C01810=1045.452,114.754,411.757,170.471,36.700,156.909
C01811=1045.446,114.505,411.777,170.469,36.699,156.908
C01812=1045.440,114.256,411.797,170.467,36.698,156.908
C01813=1045.434,114.007,411.817,170.464,36.696,156.908
C01814=1045.428,113.757,411.838,170.463,36.695,156.908
C01815=1045.422,113.509,411.858,170.461,36.693,156.907
C01816=1045.416,113.260,411.878,170.459,36.692,156.907
C01817=1045.410,113.010,411.898,170.458,36.690,156.907
C01818=1045.404,112.761,411.918,170.456,36.689,156.906
C01819=1045.398,112.512,411.937,170.453,36.687,156.906
C01820=1045.391,112.263,411.957,170.451,36.686,156.906
C01821=1045.385,112.014,411.977,170.450,36.684,156.906
C01822=1045.379,111.765,411.997,170.448,36.683,156.905
C01823=1045.373,111.515,412.018,170.446,36.681,156.905
C01824=1045.367,111.267,412.038,170.444,36.680,156.905
C01825=1045.361,111.018,412.058,170.442,36.679,156.904
C01826=1045.354,110.768,412.078,170.440,36.677,156.904
C01827=1045.348,110.519,412.097,170.438,36.676,156.904
C01828=1045.342,110.270,412.117,170.437,36.674,156.904
C01829=1045.336,110.020,412.137,170.435,36.673,156.903
C01830=1045.328,109.735,412.160,170.432,36.671,156.903
C01831=1045.322,109.449,412.183,170.430,36.669,156.903
C01832=1045.314,109.163,412.205,170.428,36.668,156.902
C01833=1045.308,108.877,412.228,170.426,36.666,156.902
C01834=1045.301,108.627,412.248,170.424,36.665,156.902
C01835=1045.295,108.379,412.268,170.423,36.664,156.902
C01836=1045.288,108.130,412.287,170.420,36.662,156.901
C01837=1045.283,107.881,412.307,170.418,36.661,156.901
C01838=1045.276,107.631,412.327,170.416,36.659,156.901
C01839=1045.270,107.382,412.347,170.415,36.658,156.900
C01840=1045.264,107.133,412.366,170.413,36.656,156.900
C01841=1045.258,106.883,412.387,170.411,36.655,156.900
C01842=1045.251,106.635,412.406,170.409,36.653,156.900
C01843=1045.245,106.386,412.425,170.407,36.652,156.899
C01844=1045.239,106.137,412.445,170.405,36.651,156.899
C01845=1045.233,105.887,412.466,170.403,36.650,156.899
C01846=1045.227,105.638,412.485,170.402,36.648,156.898
C01847=1045.221,105.389,412.505,170.399,36.646,156.898
C01848=1045.214,105.140,412.524,170.397,36.645,156.898
C01849=1045.208,104.890,412.544,170.396,36.643,156.898
C01850=1045.202,104.642,412.564,170.394,36.642,156.897
C01851=1045.196,104.392,412.583,170.392,36.641,156.897
C01852=1045.190,104.143,412.603,170.391,36.639,156.897
C01853=1045.184,103.894,412.623,170.388,36.638,156.896
C01854=1045.177,103.645,412.642,170.386,36.637,156.896
C01855=1045.171,103.396,412.662,170.384,36.635,156.896
C01856=1045.166,103.146,412.681,170.383,36.633,156.896
C01857=1045.160,102.898,412.701,170.381,36.632,156.895
C01858=1045.154,102.649,412.721,170.379,36.630,156.895
C01859=1045.147,102.399,412.741,170.377,36.629,156.895
C01860=1045.141,102.150,412.760,170.375,36.628,156.895
C01861=1045.135,101.901,412.779,170.373,36.626,156.894
C01862=1045.129,101.652,412.799,170.372,36.625,156.894
C01863=1045.123,101.402,412.818,170.370,36.624,156.894
C01864=1045.117,101.154,412.838,170.368,36.622,156.893
C01865=1045.110,100.904,412.857,170.366,36.620,156.893
C01866=1045.104,100.655,412.877,170.364,36.619,156.893
C01867=1045.098,100.406,412.897,170.362,36.618,156.893
C01868=1045.092,100.157,412.916,170.360,36.616,156.892
C01869=1045.086,99.908,412.935,170.359,36.615,156.892
C01870=1045.079,99.658,412.956,170.357,36.614,156.892
C01871=1045.073,99.409,412.974,170.354,36.612,156.892
C01872=1045.067,99.160,412.993,170.353,36.611,156.891
C01873=1045.061,98.911,413.013,170.351,36.609,156.891
C01874=1045.055,98.662,413.032,170.349,36.608,156.891
C01875=1045.048,98.413,413.051,170.348,36.607,156.890
C01876=1045.042,98.163,413.071,170.346,36.605,156.890
C01877=1045.035,97.914,413.090,170.343,36.604,156.890
C01878=1045.029,97.665,413.110,170.341,36.602,156.890
C01879=1045.024,97.416,413.129,170.340,36.601,156.889
C01880=1045.017,97.167,413.148,170.338,36.600,156.889
C01881=1045.011,96.918,413.167,170.336,36.599,156.889
C01882=1045.005,96.669,413.186,170.335,36.597,156.889
C01883=1044.999,96.418,413.206,170.332,36.596,156.888
C01884=1044.992,96.170,413.225,170.330,36.594,156.888
C01885=1044.986,95.921,413.244,170.329,36.593,156.888
C01886=1044.980,95.671,413.263,170.327,36.591,156.887
C01887=1044.974,95.423,413.283,170.325,36.590,156.887
C01888=1044.967,95.173,413.302,170.324,36.589,156.887
C01889=1044.962,94.924,413.321,170.321,36.587,156.887
C01890=1044.956,94.675,413.340,170.319,36.586,156.886
C01891=1044.949,94.426,413.359,170.318,36.584,156.886
C01892=1044.943,94.176,413.379,170.316,36.583,156.886
C01893=1044.937,93.927,413.398,170.314,36.582,156.886
C01894=1044.930,93.642,413.420,170.312,36.580,156.885
C01895=1044.923,93.355,413.441,170.309,36.579,156.885
C01896=1044.916,93.069,413.464,170.307,36.577,156.885
C01897=1044.909,92.783,413.486,170.305,36.575,156.884
C01898=1044.902,92.534,413.505,170.304,36.574,156.884
C01899=1044.896,92.285,413.525,170.302,36.572,156.884
C01900=1044.890,92.036,413.543,170.300,36.571,156.884
C01901=1044.884,91.787,413.562,170.298,36.569,156.883
C01902=1044.878,91.538,413.581,170.296,36.568,156.883
C01903=1044.872,91.288,413.600,170.294,36.567,156.883
C01904=1044.866,91.039,413.619,170.293,36.566,156.883
C01905=1044.860,90.790,413.639,170.291,36.564,156.882
C01906=1044.853,90.541,413.658,170.289,36.562,156.882
C01907=1044.848,90.292,413.677,170.287,36.561,156.882
C01908=1044.841,90.043,413.695,170.285,36.560,156.881
C01909=1044.835,89.793,413.714,170.283,36.559,156.881
C01910=1044.829,89.544,413.733,170.282,36.557,156.881
C01911=1044.822,89.294,413.752,170.280,36.556,156.881
C01912=1044.816,89.045,413.771,170.278,36.554,156.880
C01913=1044.809,88.796,413.790,170.276,36.553,156.880
C01914=1044.803,88.546,413.809,170.274,36.552,156.880
C01915=1044.797,88.297,413.828,170.272,36.551,156.880
C01916=1044.791,88.048,413.846,170.271,36.549,156.879
C01917=1044.784,87.799,413.865,170.269,36.548,156.879
C01918=1044.779,87.550,413.884,170.267,36.546,156.879
C01919=1044.772,87.301,413.903,170.265,36.545,156.879
C01920=1044.766,87.051,413.921,170.263,36.544,156.878
C01921=1044.759,86.802,413.940,170.261,36.543,156.878
C01922=1044.754,86.553,413.959,170.259,36.541,156.878
C01923=1044.747,86.304,413.978,170.258,36.540,156.878
C01924=1044.741,86.055,413.997,170.256,36.538,156.877
C01925=1044.734,85.805,414.015,170.254,36.537,156.877
C01926=1044.729,85.556,414.034,170.252,36.536,156.877
C01927=1044.722,85.307,414.053,170.250,36.534,156.877
C01928=1044.716,85.058,414.072,170.248,36.533,156.876
C01929=1044.709,84.809,414.090,170.247,36.532,156.876
C01930=1044.703,84.560,414.109,170.245,36.530,156.876
C01931=1044.697,84.310,414.128,170.243,36.529,156.876
C01932=1044.691,84.061,414.147,170.242,36.528,156.875
C01933=1044.684,83.812,414.166,170.239,36.526,156.875
C01934=1044.678,83.562,414.184,170.237,36.525,156.875
C01935=1044.673,83.313,414.203,170.236,36.524,156.875
C01936=1044.666,83.064,414.221,170.234,36.522,156.874
C01937=1044.660,82.815,414.240,170.232,36.521,156.874
C01938=1044.654,82.566,414.258,170.231,36.519,156.874
C01939=1044.647,82.317,414.277,170.228,36.518,156.873
C01940=1044.642,82.067,414.296,170.226,36.517,156.873
C01941=1044.636,81.818,414.314,170.225,36.516,156.873
C01942=1044.629,81.569,414.333,170.223,36.514,156.873
C01943=1044.623,81.320,414.351,170.221,36.513,156.872
C01944=1044.616,81.070,414.370,170.220,36.511,156.872
C01945=1044.611,80.821,414.389,170.218,36.510,156.872
C01946=1044.604,80.572,414.408,170.215,36.509,156.872
C01947=1044.598,80.322,414.426,170.214,36.507,156.871
C01948=1044.592,80.074,414.444,170.212,36.506,156.871
C01949=1044.586,79.825,414.463,170.210,36.504,156.871
C01950=1044.580,79.575,414.482,170.209,36.503,156.871
C01951=1044.574,79.325,414.500,170.207,36.502,156.870
C01952=1044.568,79.076,414.519,170.204,36.500,156.870
C01953=1044.561,78.827,414.537,170.203,36.499,156.870
C01954=1044.555,78.578,414.556,170.201,36.497,156.870
C01955=1044.549,78.328,414.574,170.199,36.496,156.869
C01956=1044.543,78.080,414.592,170.198,36.495,156.869
C01957=1044.536,77.831,414.611,170.196,36.494,156.869
C01958=1044.529,77.544,414.632,170.194,36.492,156.869
C01959=1044.523,77.258,414.653,170.191,36.491,156.868
C01960=1044.515,76.972,414.674,170.189,36.489,156.868
C01961=1044.508,76.686,414.696,170.187,36.487,156.868
C01962=1044.502,76.437,414.714,170.186,36.486,156.867
C01963=1044.496,76.188,414.732,170.184,36.485,156.867
C01964=1044.490,75.939,414.751,170.182,36.484,156.867
C01965=1044.483,75.689,414.768,170.180,36.482,156.867
C01966=1044.476,75.440,414.787,170.178,36.481,156.866
C01967=1044.470,75.191,414.805,170.176,36.479,156.866
C01968=1044.464,74.941,414.823,170.174,36.478,156.866
C01969=1044.457,74.692,414.842,170.173,36.477,156.866
C01970=1044.452,74.443,414.859,170.171,36.476,156.865
C01971=1044.445,74.194,414.878,170.169,36.474,156.865
C01972=1044.439,73.945,414.897,170.167,36.473,156.865
C01973=1044.433,73.695,414.915,170.165,36.472,156.865
C01974=1044.426,73.446,414.933,170.163,36.471,156.864
C01975=1044.420,73.196,414.951,170.162,36.469,156.864
C01976=1044.415,72.948,414.969,170.160,36.467,156.864
C01977=1044.408,72.698,414.987,170.158,36.466,156.864
C01978=1044.402,72.449,415.006,170.157,36.465,156.863
C01979=1044.395,72.199,415.023,170.154,36.464,156.863
C01980=1044.389,71.950,415.042,170.152,36.462,156.863
C01981=1044.383,71.701,415.060,170.151,36.461,156.863
C01982=1044.377,71.452,415.078,170.149,36.460,156.862
C01983=1044.371,71.202,415.096,170.147,36.459,156.862
C01984=1044.364,70.953,415.115,170.146,36.457,156.862
C01985=1044.359,70.704,415.132,170.143,36.455,156.862
C01986=1044.352,70.455,415.151,170.141,36.454,156.861
C01987=1044.346,70.205,415.169,170.140,36.453,156.861
C01988=1044.339,69.956,415.186,170.138,36.452,156.861
C01989=1044.333,69.707,415.205,170.136,36.450,156.861
C01990=1044.327,69.458,415.223,170.135,36.449,156.860
C01991=1044.321,69.209,415.241,170.133,36.448,156.860
C01992=1044.315,68.959,415.259,170.130,36.447,156.860
C01993=1044.308,68.709,415.276,170.129,36.445,156.860
C01994=1044.302,68.461,415.295,170.127,36.444,156.860
C01995=1044.296,68.211,415.313,170.125,36.443,156.859
C01996=1044.290,67.962,415.331,170.124,36.442,156.859
C01997=1044.283,67.713,415.349,170.122,36.440,156.859
C01998=1044.277,67.464,415.366,170.120,36.438,156.858
C01999=1044.271,67.214,415.384,170.117,36.437,156.858
C02000=1044.265,66.965,415.403,170.116,36.436,156.858
C02001=1044.258,66.715,415.420,170.114,36.435,156.858
C02002=1044.252,66.466,415.438,170.112,36.433,156.857
C02003=1044.246,66.217,415.456,170.111,36.432,156.857
C02004=1044.240,65.968,415.474,170.109,36.431,156.857
C02005=1044.233,65.718,415.492,170.107,36.430,156.857
C02006=1044.227,65.469,415.509,170.105,36.428,156.857
C02007=1044.221,65.220,415.528,170.103,36.427,156.856
C02008=1044.214,64.970,415.545,170.101,36.426,156.856
C02009=1044.209,64.721,415.563,170.100,36.425,156.856
C02010=1044.202,64.472,415.581,170.098,36.423,156.856
C02011=1044.195,64.223,415.599,170.096,36.422,156.855
C02012=1044.189,63.973,415.617,170.095,36.421,156.855
C02013=1044.184,63.724,415.634,170.093,36.420,156.855
C02014=1044.177,63.475,415.652,170.090,36.418,156.855
C02015=1044.170,63.225,415.669,170.088,36.417,156.854
C02016=1044.164,62.976,415.687,170.087,36.416,156.854
C02017=1044.157,62.727,415.705,170.085,36.415,156.854
C02018=1044.151,62.478,415.722,170.083,36.413,156.854
C02019=1044.144,62.228,415.740,170.082,36.412,156.853
C02020=1044.139,61.979,415.757,170.080,36.411,156.853
C02021=1044.132,61.730,415.775,170.078,36.410,156.853
C02022=1044.124,61.443,415.795,170.075,36.408,156.853
C02023=1044.117,61.157,415.815,170.073,36.407,156.853
C02024=1044.110,60.871,415.835,170.071,36.406,156.852
C02025=1044.103,60.585,415.855,170.069,36.404,156.852
C02026=1044.096,60.335,415.873,170.068,36.403,156.852
C02027=1044.090,60.085,415.890,170.066,36.402,156.852
C02028=1044.083,59.837,415.908,170.063,36.401,156.851
C02029=1044.076,59.588,415.926,170.062,36.399,156.851
C02030=1044.070,59.338,415.943,170.060,36.398,156.851
C02031=1044.064,59.089,415.960,170.058,36.397,156.851
C02032=1044.058,58.840,415.978,170.056,36.396,156.850
C02033=1044.051,58.590,415.996,170.055,36.394,156.850
C02034=1044.045,58.342,416.013,170.053,36.393,156.850
C02035=1044.039,58.092,416.031,170.051,36.392,156.850
C02036=1044.032,57.843,416.048,170.049,36.391,156.849
C02037=1044.026,57.593,416.066,170.047,36.389,156.849
C02038=1044.019,57.344,416.083,170.045,36.388,156.849
C02039=1044.013,57.095,416.100,170.043,36.387,156.849
C02040=1044.007,56.845,416.118,170.042,36.386,156.849
C02041=1044.000,56.596,416.135,170.040,36.385,156.848
C02042=1043.995,56.346,416.152,170.038,36.384,156.848
C02043=1043.988,56.097,416.169,170.037,36.382,156.848
C02044=1043.982,55.848,416.186,170.034,36.381,156.848
C02045=1043.976,55.598,416.204,170.032,36.380,156.848
C02046=1043.969,55.349,416.222,170.031,36.379,156.847
C02047=1043.963,55.100,416.239,170.029,36.377,156.847
C02048=1043.957,54.851,416.256,170.027,36.376,156.847
C02049=1043.950,54.602,416.273,170.025,36.375,156.847
C02050=1043.944,54.352,416.291,170.024,36.373,156.846
C02051=1043.937,54.103,416.309,170.021,36.372,156.846
C02052=1043.931,53.854,416.326,170.019,36.371,156.846
C02053=1043.925,53.604,416.343,170.018,36.370,156.846
C02054=1043.919,53.355,416.360,170.016,36.368,156.845
C02055=1043.913,53.105,416.378,170.014,36.367,156.845
C02056=1043.907,52.856,416.395,170.012,36.366,156.845
C02057=1043.900,52.607,416.412,170.011,36.365,156.845
C02058=1043.894,52.358,416.430,170.009,36.363,156.844
C02059=1043.888,52.108,416.446,170.006,36.362,156.844
C02060=1043.881,51.859,416.463,170.005,36.361,156.844
C02061=1043.875,51.609,416.481,170.003,36.360,156.844
C02062=1043.869,51.361,416.498,170.001,36.358,156.844
C02063=1043.862,51.111,416.515,170.000,36.357,156.843
C02064=1043.857,50.862,416.532,169.998,36.356,156.843
C02065=1043.850,50.612,416.550,169.996,36.355,156.843
C02066=1043.844,50.363,416.567,169.993,36.353,156.843
C02067=1043.838,50.114,416.585,169.992,36.352,156.842
C02068=1043.831,49.865,416.602,169.990,36.351,156.842
C02069=1043.825,49.615,416.618,169.988,36.349,156.842
C02070=1043.819,49.366,416.636,169.987,36.348,156.842
C02071=1043.813,49.116,416.653,169.985,36.347,156.841
C02072=1043.807,48.867,416.671,169.983,36.346,156.841
C02073=1043.800,48.617,416.687,169.981,36.344,156.841
C02074=1043.794,48.369,416.704,169.979,36.343,156.841
C02075=1043.788,48.119,416.722,169.977,36.342,156.840
C02076=1043.782,47.869,416.738,169.975,36.341,156.840
C02077=1043.775,47.620,416.756,169.974,36.339,156.840
C02078=1043.770,47.371,416.773,169.972,36.338,156.840
C02079=1043.763,47.121,416.790,169.970,36.337,156.840
C02080=1043.757,46.872,416.807,169.969,36.336,156.839
C02081=1043.751,46.624,416.824,169.966,36.334,156.839
C02082=1043.745,46.373,416.841,169.964,36.333,156.839
C02083=1043.739,46.124,416.858,169.963,36.332,156.839
C02084=1043.732,45.875,416.875,169.961,36.330,156.838
C02085=1043.727,45.625,416.892,169.959,36.329,156.838
C02086=1043.720,45.339,416.912,169.957,36.328,156.838
C02087=1043.712,45.052,416.932,169.955,36.326,156.838
C02088=1043.705,44.766,416.950,169.952,36.325,156.837
C02089=1043.698,44.480,416.970,169.950,36.323,156.837
C02090=1043.692,44.230,416.988,169.949,36.322,156.837
C02091=1043.686,43.981,417.005,169.947,36.321,156.837
C02092=1043.679,43.731,417.022,169.945,36.320,156.836
C02093=1043.674,43.482,417.039,169.944,36.318,156.836
C02094=1043.668,43.233,417.056,169.942,36.317,156.836
C02095=1043.661,42.983,417.072,169.940,36.316,156.836
C02096=1043.655,42.734,417.089,169.937,36.315,156.835
C02097=1043.648,42.484,417.106,169.936,36.313,156.835
C02098=1043.642,42.235,417.123,169.934,36.312,156.835
C02099=1043.636,41.986,417.139,169.932,36.311,156.835
C02100=1043.629,41.737,417.157,169.930,36.309,156.835
C02101=1043.623,41.487,417.173,169.929,36.308,156.834
C02102=1043.616,41.238,417.190,169.927,36.307,156.834
C02103=1043.610,40.989,417.206,169.925,36.306,156.834
C02104=1043.604,40.739,417.223,169.923,36.305,156.834
C02105=1043.598,40.490,417.240,169.921,36.304,156.833
C02106=1043.592,40.240,417.256,169.919,36.302,156.833
C02107=1043.586,39.991,417.274,169.917,36.301,156.833
C02108=1043.580,39.741,417.290,169.916,36.300,156.833
C02109=1043.573,39.493,417.307,169.914,36.299,156.833
C02110=1043.567,39.243,417.324,169.912,36.297,156.832
C02111=1043.561,38.993,417.340,169.909,36.296,156.832
C02112=1043.555,38.744,417.357,169.908,36.295,156.832
C02113=1043.549,38.495,417.374,169.906,36.294,156.832
C02114=1043.542,38.245,417.390,169.904,36.293,156.832
C02115=1043.536,37.996,417.407,169.903,36.292,156.831
C02116=1043.530,37.747,417.423,169.901,36.290,156.831
C02117=1043.523,37.497,417.440,169.899,36.289,156.831
C02118=1043.517,37.248,417.457,169.897,36.288,156.831
C02119=1043.510,36.998,417.474,169.896,36.287,156.830
C02120=1043.505,36.749,417.490,169.893,36.285,156.830
C02121=1043.498,36.500,417.506,169.891,36.285,156.830
C02122=1043.491,36.250,417.523,169.889,36.283,156.830
C02123=1043.485,36.001,417.539,169.888,36.282,156.830
C02124=1043.479,35.752,417.555,169.886,36.281,156.829
C02125=1043.472,35.502,417.573,169.884,36.280,156.829
C02126=1043.466,35.253,417.589,169.882,36.279,156.829
C02127=1043.460,35.004,417.605,169.880,36.278,156.829
C02128=1043.453,34.754,417.621,169.878,36.276,156.829
C02129=1043.447,34.504,417.638,169.876,36.275,156.828
C02130=1043.441,34.256,417.654,169.874,36.274,156.828
C02131=1043.435,34.006,417.671,169.872,36.273,156.828
C02132=1043.428,33.757,417.687,169.871,36.272,156.828
C02133=1043.422,33.507,417.703,169.869,36.271,156.827
C02134=1043.416,33.258,417.719,169.867,36.269,156.827
C02135=1043.409,33.009,417.737,169.865,36.268,156.827
C02136=1043.403,32.759,417.753,169.864,36.267,156.827
C02137=1043.397,32.510,417.769,169.861,36.266,156.827
C02138=1043.390,32.261,417.785,169.859,36.265,156.826
C02139=1043.384,32.011,417.801,169.857,36.264,156.826
C02140=1043.378,31.761,417.818,169.856,36.262,156.826
C02141=1043.371,31.513,417.835,169.854,36.261,156.826
C02142=1043.365,31.263,417.851,169.852,36.260,156.825
C02143=1043.358,31.014,417.867,169.850,36.259,156.825
C02144=1043.352,30.764,417.883,169.849,36.258,156.825
C02145=1043.346,30.515,417.899,169.846,36.257,156.825
C02146=1043.340,30.266,417.916,169.844,36.255,156.825
C02147=1043.334,30.015,417.932,169.842,36.254,156.824
C02148=1043.327,29.766,417.948,169.840,36.253,156.824
C02149=1043.321,29.517,417.964,169.839,36.252,156.824
C02150=1043.314,29.231,417.983,169.837,36.251,156.824
C02151=1043.307,28.944,418.002,169.835,36.249,156.824
C02152=1043.300,28.657,418.020,169.833,36.248,156.823
C02153=1043.292,28.370,418.039,169.830,36.246,156.823
C02154=1043.286,28.121,418.055,169.828,36.245,156.823
C02155=1043.279,27.872,418.071,169.826,36.244,156.823
C02156=1043.273,27.623,418.087,169.824,36.243,156.823
C02157=1043.267,27.373,418.103,169.822,36.242,156.822
C02158=1043.260,27.124,418.120,169.821,36.241,156.822
C02159=1043.254,26.874,418.136,169.819,36.240,156.822
C02160=1043.248,26.625,418.152,169.817,36.239,156.822
C02161=1043.242,26.376,418.168,169.815,36.237,156.821
C02162=1043.236,26.127,418.184,169.813,36.236,156.821
C02163=1043.228,25.877,418.200,169.811,36.236,156.821
C02164=1043.222,25.627,418.216,169.809,36.234,156.821
C02165=1043.216,25.378,418.232,169.807,36.233,156.821
C02166=1043.210,25.128,418.247,169.805,36.232,156.821
C02167=1043.204,24.879,418.264,169.804,36.231,156.820
C02168=1043.197,24.629,418.280,169.802,36.230,156.820
C02169=1043.191,24.380,418.296,169.800,36.228,156.820
C02170=1043.184,24.131,418.312,169.798,36.228,156.820
C02171=1043.178,23.882,418.328,169.795,36.227,156.820
C02172=1043.172,23.632,418.344,169.794,36.225,156.819
C02173=1043.166,23.383,418.359,169.792,36.224,156.819
C02174=1043.159,23.133,418.376,169.790,36.223,156.819
C02175=1043.153,22.884,418.391,169.788,36.222,156.819
C02176=1043.147,22.634,418.408,169.786,36.221,156.818
C02177=1043.140,22.385,418.423,169.785,36.219,156.818
C02178=1043.134,22.136,418.440,169.783,36.219,156.818
C02179=1043.128,21.886,418.454,169.781,36.218,156.818
C02180=1043.122,21.637,418.471,169.778,36.216,156.818
C02181=1043.115,21.388,418.486,169.776,36.215,156.817
C02182=1043.109,21.138,418.503,169.775,36.214,156.817
C02183=1043.103,20.888,418.519,169.773,36.213,156.817
C02184=1043.096,20.639,418.534,169.771,36.212,156.817
C02185=1043.090,20.389,418.550,169.769,36.211,156.817
C02186=1043.084,20.140,418.566,169.767,36.210,156.817
C02187=1043.078,19.890,418.582,169.766,36.209,156.816
C02188=1043.071,19.641,418.597,169.764,36.207,156.816
C02189=1043.065,19.392,418.614,169.762,36.207,156.816
C02190=1043.059,19.143,418.629,169.759,36.205,156.816
C02191=1043.052,18.893,418.644,169.757,36.204,156.815
C02192=1043.046,18.644,418.660,169.755,36.203,156.815
C02193=1043.039,18.394,418.677,169.754,36.202,156.815
C02194=1043.033,18.144,418.692,169.752,36.201,156.815
C02195=1043.027,17.895,418.708,169.750,36.200,156.815
C02196=1043.020,17.646,418.723,169.748,36.199,156.815
C02197=1043.014,17.396,418.739,169.746,36.198,156.814
C02198=1043.008,17.147,418.755,169.745,36.197,156.814
C02199=1043.002,16.897,418.770,169.742,36.196,156.814
C02200=1042.995,16.648,418.786,169.740,36.194,156.814
C02201=1042.989,16.399,418.801,169.738,36.194,156.814
C02202=1042.983,16.149,418.817,169.736,36.193,156.813
C02203=1042.976,15.900,418.833,169.734,36.191,156.813
C02204=1042.970,15.650,418.848,169.733,36.190,156.813
C02205=1042.964,15.401,418.864,169.731,36.189,156.813
C02206=1042.957,15.152,418.880,169.729,36.188,156.813
C02207=1042.952,14.902,418.895,169.727,36.187,156.812
C02208=1042.945,14.653,418.911,169.725,36.186,156.812
C02209=1042.938,14.403,418.926,169.722,36.185,156.812
C02210=1042.933,14.154,418.942,169.721,36.184,156.812
C02211=1042.926,13.904,418.957,169.719,36.183,156.812
C02212=1042.919,13.655,418.973,169.717,36.182,156.811
C02213=1042.913,13.406,418.987,169.715,36.181,156.811
C02214=1042.906,13.120,419.005,169.713,36.180,156.811
C02215=1042.898,12.835,419.023,169.711,36.178,156.811
C02216=1042.891,12.550,419.041,169.709,36.177,156.811
C02217=1042.884,12.265,419.059,169.707,36.176,156.811
C02218=1042.877,12.015,419.074,169.704,36.175,156.810
C02219=1042.871,11.765,419.089,169.702,36.174,156.810
C02220=1042.864,11.516,419.104,169.700,36.173,156.810
C02221=1042.858,11.267,419.119,169.698,36.172,156.810
C02222=1042.851,11.017,419.135,169.696,36.171,156.810
C02223=1042.845,10.768,419.150,169.694,36.170,156.809
C02224=1042.839,10.518,419.165,169.692,36.169,156.809
C02225=1042.832,10.269,419.181,169.691,36.168,156.809
C02226=1042.826,10.019,419.196,169.689,36.167,156.809
C02227=1042.819,9.770,419.212,169.687,36.166,156.809
C02228=1042.813,9.520,419.227,169.685,36.165,156.809
C02229=1042.807,9.271,419.242,169.682,36.164,156.808
C02230=1042.800,9.022,419.257,169.680,36.163,156.808
C02231=1042.793,8.772,419.272,169.678,36.162,156.808
C02232=1042.788,8.522,419.288,169.676,36.161,156.808
C02233=1042.781,8.273,419.303,169.675,36.160,156.808
C02234=1042.775,8.023,419.318,169.673,36.159,156.808
C02235=1042.768,7.774,419.333,169.671,36.158,156.807
C02236=1042.762,7.524,419.348,169.669,36.157,156.807
C02237=1042.755,7.275,419.364,169.667,36.156,156.807
C02238=1042.750,7.026,419.378,169.665,36.155,156.807
C02239=1042.743,6.776,419.393,169.662,36.154,156.807
C02240=1042.736,6.527,419.409,169.660,36.153,156.807
C02241=1042.730,6.278,419.424,169.659,36.152,156.806
C02242=1042.724,6.028,419.440,169.657,36.151,156.806
C02243=1042.718,5.778,419.455,169.655,36.150,156.806
C02244=1042.712,5.528,419.469,169.653,36.149,156.806
C02245=1042.705,5.279,419.485,169.651,36.148,156.806
C02246=1042.699,5.030,419.500,169.649,36.147,156.805
C02247=1042.693,4.781,419.515,169.647,36.146,156.805
C02248=1042.686,4.531,419.530,169.645,36.145,156.805
C02249=1042.680,4.282,419.545,169.643,36.144,156.805
C02250=1042.673,4.033,419.560,169.641,36.143,156.805
C02251=1042.667,3.783,419.575,169.639,36.142,156.805
C02252=1042.661,3.533,419.590,169.637,36.141,156.804
C02253=1042.655,3.283,419.606,169.635,36.140,156.804
C02254=1042.649,3.034,419.620,169.633,36.139,156.804
C02255=1042.642,2.785,419.636,169.631,36.138,156.804
C02256=1042.636,2.536,419.651,169.629,36.137,156.804
C02257=1042.630,2.286,419.666,169.627,36.136,156.803
C02258=1042.623,2.036,419.681,169.625,36.135,156.803
C02259=1042.617,1.787,419.696,169.624,36.134,156.803
C02260=1042.611,1.538,419.710,169.622,36.133,156.803
C02261=1042.605,1.288,419.725,169.619,36.132,156.803
C02262=1042.598,1.038,419.740,169.617,36.131,156.803
C02263=1042.592,0.789,419.755,169.615,36.130,156.802
C02264=1042.585,0.540,419.771,169.613,36.129,156.802
C02265=1042.580,0.291,419.785,169.611,36.128,156.802
C02266=1042.573,0.041,419.800,169.609,36.127,156.802
C02267=1042.567,-0.209,419.815,169.607,36.126,156.802
C02268=1042.560,-0.458,419.830,169.605,36.125,156.802
C02269=1042.555,-0.707,419.845,169.604,36.124,156.801
C02270=1042.548,-0.957,419.860,169.602,36.123,156.801
C02271=1042.543,-1.207,419.875,169.599,36.121,156.801
C02272=1042.536,-1.457,419.890,169.597,36.121,156.801
C02273=1042.530,-1.705,419.905,169.595,36.120,156.801
C02274=1042.524,-1.955,419.920,169.593,36.119,156.801
C02275=1042.518,-2.205,419.935,169.591,36.118,156.800
C02276=1042.511,-2.454,419.950,169.589,36.117,156.800
C02277=1042.505,-2.703,419.964,169.587,36.116,156.800
C02278=1042.498,-2.987,419.981,169.585,36.114,156.800
C02279=1042.490,-3.270,419.998,169.583,36.113,156.799
C02280=1042.484,-3.554,420.015,169.581,36.112,156.799
C02281=1042.477,-3.838,420.031,169.578,36.111,156.799
C02282=1042.470,-4.087,420.046,169.576,36.110,156.799
C02283=1042.464,-4.336,420.060,169.574,36.109,156.799
C02284=1042.458,-4.586,420.075,169.572,36.108,156.799
C02285=1042.451,-4.835,420.090,169.570,36.108,156.799
C02286=1042.444,-5.085,420.104,169.568,36.106,156.798
C02287=1042.439,-5.334,420.118,169.566,36.106,156.798
C02288=1042.432,-5.584,420.133,169.564,36.105,156.798
C02289=1042.425,-5.833,420.148,169.562,36.104,156.798
C02290=1042.419,-6.083,420.163,169.560,36.103,156.798
C02291=1042.413,-6.332,420.177,169.558,36.102,156.798
C02292=1042.407,-6.582,420.192,169.556,36.101,156.797
C02293=1042.400,-6.831,420.206,169.554,36.101,156.797
C02294=1042.393,-7.081,420.221,169.551,36.099,156.797
C02295=1042.388,-7.330,420.235,169.549,36.099,156.797
C02296=1042.381,-7.579,420.250,169.547,36.097,156.797
C02297=1042.375,-7.830,420.264,169.545,36.097,156.797
C02298=1042.369,-8.079,420.278,169.543,36.096,156.797
C02299=1042.362,-8.328,420.293,169.541,36.095,156.796
C02300=1042.355,-8.578,420.308,169.539,36.094,156.796
C02301=1042.350,-8.827,420.322,169.537,36.093,156.796
C02302=1042.343,-9.077,420.337,169.535,36.092,156.796
C02303=1042.336,-9.326,420.351,169.533,36.091,156.796
C02304=1042.330,-9.575,420.365,169.531,36.090,156.796
C02305=1042.324,-9.825,420.380,169.530,36.090,156.795
C02306=1042.317,-10.075,420.394,169.527,36.089,156.795
C02307=1042.311,-10.324,420.409,169.525,36.088,156.795
C02308=1042.305,-10.574,420.423,169.523,36.087,156.795
C02309=1042.298,-10.823,420.437,169.521,36.086,156.795
C02310=1042.292,-11.072,420.452,169.519,36.085,156.795
C02311=1042.286,-11.323,420.466,169.517,36.084,156.795
C02312=1042.280,-11.571,420.480,169.515,36.083,156.794
C02313=1042.274,-11.821,420.495,169.513,36.082,156.794
C02314=1042.267,-12.071,420.509,169.511,36.082,156.794
C02315=1042.261,-12.320,420.523,169.509,36.080,156.794
C02316=1042.255,-12.570,420.537,169.507,36.080,156.794
C02317=1042.248,-12.820,420.552,169.505,36.079,156.794
C02318=1042.242,-13.068,420.566,169.502,36.078,156.793
C02319=1042.236,-13.319,420.581,169.500,36.077,156.793
C02320=1042.230,-13.568,420.595,169.498,36.076,156.793
C02321=1042.223,-13.818,420.609,169.496,36.075,156.793
C02322=1042.217,-14.067,420.623,169.494,36.074,156.793
C02323=1042.211,-14.317,420.638,169.492,36.073,156.793
C02324=1042.204,-14.566,420.652,169.490,36.073,156.793
C02325=1042.199,-14.815,420.666,169.488,36.072,156.792
C02326=1042.192,-15.065,420.681,169.486,36.071,156.792
C02327=1042.186,-15.314,420.695,169.484,36.070,156.792
C02328=1042.180,-15.564,420.709,169.482,36.069,156.792
C02329=1042.173,-15.813,420.723,169.480,36.068,156.792
C02330=1042.167,-16.063,420.737,169.478,36.067,156.792
C02331=1042.160,-16.313,420.751,169.476,36.067,156.792
C02332=1042.155,-16.562,420.765,169.473,36.066,156.791
C02333=1042.148,-16.812,420.779,169.471,36.065,156.791
C02334=1042.141,-17.061,420.793,169.469,36.064,156.791
C02335=1042.135,-17.311,420.807,169.467,36.063,156.791
C02336=1042.129,-17.560,420.821,169.465,36.063,156.791
C02337=1042.123,-17.810,420.835,169.463,36.062,156.791
C02338=1042.116,-18.060,420.849,169.461,36.061,156.791
C02339=1042.109,-18.309,420.863,169.459,36.060,156.790
C02340=1042.103,-18.559,420.877,169.457,36.059,156.790
C02341=1042.097,-18.808,420.891,169.455,36.059,156.790
C02342=1042.089,-19.090,420.907,169.452,36.057,156.790
C02343=1042.083,-19.371,420.922,169.450,36.057,156.790
C02344=1042.075,-19.654,420.938,169.448,36.056,156.790
C02345=1042.069,-19.936,420.954,169.444,36.055,156.790
C02346=1042.062,-20.185,420.968,169.442,36.054,156.789
C02347=1042.055,-20.434,420.982,169.440,36.053,156.789
C02348=1042.050,-20.684,420.996,169.438,36.053,156.789
C02349=1042.043,-20.934,421.010,169.436,36.051,156.789
C02350=1042.036,-21.182,421.024,169.434,36.051,156.789
C02351=1042.030,-21.433,421.038,169.432,36.050,156.789
C02352=1042.024,-21.682,421.051,169.430,36.049,156.789
C02353=1042.018,-21.932,421.066,169.428,36.049,156.789
C02354=1042.012,-22.181,421.079,169.426,36.048,156.788
C02355=1042.005,-22.430,421.093,169.424,36.047,156.788
C02356=1041.999,-22.680,421.107,169.422,36.046,156.788
C02357=1041.993,-22.929,421.121,169.420,36.046,156.788
C02358=1041.987,-23.179,421.135,169.418,36.045,156.788
C02359=1041.980,-23.429,421.148,169.416,36.044,156.788
C02360=1041.974,-23.679,421.162,169.413,36.043,156.788
C02361=1041.968,-23.928,421.176,169.411,36.042,156.788
C02362=1041.962,-24.177,421.190,169.409,36.042,156.787
C02363=1041.955,-24.427,421.203,169.407,36.041,156.787
C02364=1041.949,-24.676,421.217,169.404,36.040,156.787
C02365=1041.942,-24.926,421.231,169.402,36.039,156.787
C02366=1041.936,-25.176,421.244,169.400,36.038,156.787
C02367=1041.930,-25.425,421.259,169.398,36.038,156.787
C02368=1041.924,-25.675,421.272,169.396,36.036,156.787
C02369=1041.918,-25.924,421.286,169.394,36.036,156.786
C02370=1041.911,-26.174,421.300,169.392,36.035,156.786
C02371=1041.905,-26.423,421.313,169.390,36.034,156.786
C02372=1041.900,-26.673,421.327,169.388,36.034,156.786
C02373=1041.893,-26.923,421.341,169.386,36.032,156.786
C02374=1041.887,-27.172,421.354,169.383,36.032,156.786
C02375=1041.880,-27.422,421.368,169.381,36.031,156.786
C02376=1041.873,-27.671,421.382,169.379,36.030,156.786
C02377=1041.867,-27.920,421.395,169.377,36.030,156.785
C02378=1041.861,-28.170,421.409,169.374,36.029,156.785
C02379=1041.855,-28.420,421.422,169.372,36.028,156.785
C02380=1041.849,-28.669,421.436,169.370,36.028,156.785
C02381=1041.842,-28.919,421.449,169.368,36.027,156.785
C02382=1041.836,-29.168,421.463,169.366,36.026,156.785
C02383=1041.829,-29.418,421.476,169.364,36.026,156.785
C02384=1041.823,-29.667,421.489,169.362,36.025,156.785
C02385=1041.816,-29.917,421.503,169.360,36.024,156.785
C02386=1041.810,-30.166,421.516,169.358,36.024,156.784
C02387=1041.804,-30.416,421.530,169.355,36.023,156.784
C02388=1041.798,-30.666,421.543,169.353,36.022,156.784
C02389=1041.791,-30.916,421.556,169.351,36.022,156.784
C02390=1041.785,-31.165,421.570,169.349,36.021,156.784
C02391=1041.779,-31.414,421.583,169.347,36.020,156.784
C02392=1041.772,-31.664,421.597,169.344,36.020,156.784
C02393=1041.766,-31.914,421.610,169.342,36.019,156.784
C02394=1041.760,-32.163,421.623,169.340,36.018,156.784
C02395=1041.753,-32.413,421.637,169.338,36.018,156.783
C02396=1041.747,-32.662,421.650,169.335,36.017,156.783
C02397=1041.740,-32.911,421.663,169.333,36.016,156.783
C02398=1041.734,-33.161,421.677,169.331,36.015,156.783
C02399=1041.728,-33.412,421.690,169.329,36.014,156.783
C02400=1041.722,-33.661,421.703,169.327,36.014,156.783
C02401=1041.716,-33.910,421.717,169.325,36.013,156.783
C02402=1041.709,-34.160,421.730,169.323,36.012,156.783
C02403=1041.703,-34.409,421.743,169.321,36.012,156.782
C02404=1041.697,-34.659,421.757,169.318,36.011,156.782
C02405=1041.691,-34.909,421.769,169.316,36.010,156.782
C02406=1041.683,-35.189,421.784,169.314,36.010,156.782
C02407=1041.677,-35.471,421.799,169.312,36.009,156.782
C02408=1041.669,-35.751,421.814,169.309,36.008,156.782
C02409=1041.663,-36.033,421.829,169.306,36.008,156.782
C02410=1041.657,-36.282,421.843,169.304,36.007,156.782
C02411=1041.650,-36.531,421.856,169.301,36.006,156.782
C02412=1041.644,-36.781,421.869,169.299,36.006,156.782
C02413=1041.637,-37.031,421.883,169.297,36.005,156.781
C02414=1041.632,-37.280,421.895,169.295,36.004,156.781
C02415=1041.625,-37.530,421.909,169.293,36.004,156.781
C02416=1041.619,-37.779,421.922,169.291,36.003,156.781
C02417=1041.613,-38.030,421.935,169.289,36.002,156.781
C02418=1041.606,-38.279,421.948,169.287,36.002,156.781
C02419=1041.600,-38.528,421.961,169.284,36.001,156.781
C02420=1041.594,-38.778,421.974,169.282,36.000,156.781
C02421=1041.588,-39.027,421.987,169.280,36.000,156.781
C02422=1041.581,-39.277,422.001,169.278,35.999,156.780
C02423=1041.575,-39.527,422.013,169.276,35.998,156.780
C02424=1041.568,-39.776,422.026,169.274,35.998,156.780
C02425=1041.562,-40.025,422.039,169.271,35.997,156.780
C02426=1041.556,-40.275,422.052,169.269,35.997,156.780
C02427=1041.549,-40.525,422.065,169.267,35.996,156.780
C02428=1041.543,-40.775,422.077,169.265,35.996,156.780
C02429=1041.537,-41.024,422.091,169.262,35.995,156.780
C02430=1041.530,-41.273,422.104,169.259,35.994,156.780
C02431=1041.524,-41.523,422.116,169.257,35.994,156.780
C02432=1041.518,-41.772,422.130,169.255,35.993,156.780
C02433=1041.511,-42.023,422.142,169.253,35.993,156.780
C02434=1041.505,-42.272,422.155,169.251,35.992,156.779
C02435=1041.499,-42.522,422.168,169.249,35.991,156.779
C02436=1041.493,-42.771,422.181,169.246,35.991,156.779
C02437=1041.487,-43.021,422.194,169.244,35.990,156.779
C02438=1041.480,-43.270,422.206,169.242,35.990,156.779
C02439=1041.474,-43.520,422.219,169.240,35.989,156.779
C02440=1041.468,-43.769,422.232,169.238,35.989,156.779
C02441=1041.461,-44.020,422.245,169.235,35.988,156.779
C02442=1041.455,-44.269,422.258,169.233,35.987,156.779
C02443=1041.448,-44.519,422.270,169.231,35.987,156.779
C02444=1041.442,-44.768,422.284,169.229,35.987,156.779
C02445=1041.436,-45.018,422.296,169.227,35.986,156.778
C02446=1041.430,-45.267,422.309,169.224,35.985,156.778
C02447=1041.423,-45.516,422.321,169.222,35.985,156.778
C02448=1041.417,-45.766,422.334,169.220,35.984,156.778
C02449=1041.411,-46.016,422.347,169.218,35.983,156.778
C02450=1041.405,-46.266,422.360,169.216,35.983,156.778
C02451=1041.398,-46.514,422.372,169.213,35.983,156.778
C02452=1041.392,-46.764,422.385,169.210,35.982,156.778
C02453=1041.386,-47.014,422.398,169.208,35.981,156.778
C02454=1041.380,-47.264,422.411,169.206,35.981,156.778
C02455=1041.374,-47.513,422.423,169.204,35.981,156.778
C02456=1041.368,-47.763,422.435,169.201,35.980,156.778
C02457=1041.361,-48.013,422.449,169.199,35.979,156.777
C02458=1041.355,-48.263,422.462,169.197,35.979,156.777
C02459=1041.348,-48.512,422.474,169.195,35.978,156.777
C02460=1041.342,-48.762,422.487,169.193,35.978,156.777
C02461=1041.336,-49.012,422.499,169.190,35.977,156.777
C02462=1041.330,-49.261,422.512,169.188,35.977,156.777
C02463=1041.323,-49.510,422.525,169.186,35.976,156.777
C02464=1041.318,-49.760,422.537,169.184,35.975,156.777
C02465=1041.312,-50.009,422.549,169.181,35.975,156.777
C02466=1041.306,-50.259,422.563,169.179,35.974,156.777
C02467=1041.299,-50.508,422.575,169.177,35.974,156.777
C02468=1041.293,-50.759,422.587,169.175,35.974,156.777
C02469=1041.286,-51.008,422.599,169.173,35.973,156.776
C02470=1041.279,-51.289,422.613,169.170,35.972,156.776
C02471=1041.272,-51.571,422.627,169.167,35.972,156.776
C02472=1041.264,-51.852,422.641,169.165,35.972,156.776
C02473=1041.257,-52.134,422.655,169.162,35.971,156.776
C02474=1041.251,-52.384,422.668,169.160,35.971,156.776
C02475=1041.244,-52.633,422.680,169.158,35.970,156.776
C02476=1041.238,-52.883,422.692,169.155,35.970,156.776
C02477=1041.232,-53.133,422.704,169.153,35.970,156.776
C02478=1041.225,-53.382,422.716,169.151,35.970,156.776
C02479=1041.219,-53.632,422.729,169.148,35.969,156.776
C02480=1041.213,-53.882,422.741,169.145,35.969,156.776
C02481=1041.206,-54.131,422.753,169.143,35.968,156.776
C02482=1041.200,-54.381,422.765,169.141,35.968,156.776
C02483=1041.194,-54.630,422.777,169.139,35.967,156.776
C02484=1041.187,-54.880,422.789,169.136,35.967,156.776
C02485=1041.181,-55.129,422.802,169.134,35.967,156.776
C02486=1041.174,-55.378,422.814,169.132,35.966,156.775
C02487=1041.169,-55.628,422.827,169.129,35.966,156.775
C02488=1041.162,-55.878,422.839,169.127,35.965,156.775
C02489=1041.155,-56.127,422.851,169.125,35.965,156.775
C02490=1041.149,-56.377,422.863,169.123,35.965,156.775
C02491=1041.143,-56.627,422.875,169.120,35.965,156.775
C02492=1041.136,-56.876,422.887,169.118,35.964,156.775
C02493=1041.130,-57.126,422.900,169.116,35.964,156.775
C02494=1041.123,-57.376,422.912,169.113,35.963,156.775
C02495=1041.117,-57.625,422.924,169.111,35.963,156.775
C02496=1041.112,-57.875,422.936,169.109,35.963,156.775
C02497=1041.105,-58.124,422.948,169.107,35.963,156.775
C02498=1041.099,-58.374,422.959,169.104,35.962,156.775
C02499=1041.093,-58.624,422.972,169.102,35.962,156.775
C02500=1041.086,-58.874,422.984,169.100,35.961,156.775
C02501=1041.079,-59.123,422.996,169.097,35.961,156.775
C02502=1041.073,-59.373,423.008,169.095,35.960,156.775
C02503=1041.067,-59.623,423.020,169.093,35.960,156.775
C02504=1041.061,-59.872,423.032,169.090,35.960,156.775
C02505=1041.055,-60.122,423.044,169.088,35.960,156.775
C02506=1041.048,-60.371,423.056,169.086,35.959,156.774
C02507=1041.042,-60.621,423.068,169.084,35.959,156.775
C02508=1041.036,-60.871,423.080,169.081,35.958,156.774
C02509=1041.030,-61.120,423.092,169.079,35.958,156.774
C02510=1041.023,-61.370,423.103,169.077,35.958,156.774
C02511=1041.017,-61.620,423.116,169.074,35.958,156.774
C02512=1041.011,-61.869,423.128,169.072,35.957,156.774
C02513=1041.004,-62.119,423.140,169.070,35.957,156.774
C02514=1040.999,-62.369,423.151,169.067,35.957,156.774
C02515=1040.992,-62.618,423.163,169.065,35.956,156.774
C02516=1040.986,-62.868,423.175,169.063,35.956,156.774
C02517=1040.980,-63.118,423.188,169.060,35.955,156.774
C02518=1040.973,-63.367,423.200,169.058,35.955,156.774
C02519=1040.967,-63.617,423.211,169.056,35.955,156.774
C02520=1040.961,-63.866,423.223,169.054,35.955,156.774
C02521=1040.955,-64.116,423.235,169.050,35.954,156.774
C02522=1040.948,-64.366,423.247,169.048,35.954,156.774
C02523=1040.943,-64.615,423.258,169.046,35.953,156.774
C02524=1040.937,-64.865,423.271,169.043,35.953,156.774
C02525=1040.930,-65.115,423.283,169.041,35.953,156.774
C02526=1040.924,-65.363,423.294,169.039,35.953,156.774
C02527=1040.918,-65.614,423.305,169.036,35.952,156.774
C02528=1040.912,-65.864,423.318,169.034,35.952,156.774
C02529=1040.905,-66.113,423.330,169.032,35.952,156.774
C02530=1040.899,-66.363,423.341,169.029,35.951,156.773
C02531=1040.893,-66.613,423.353,169.027,35.951,156.773
C02532=1040.887,-66.862,423.365,169.025,35.950,156.773
C02533=1040.881,-67.112,423.376,169.022,35.950,156.773
C02534=1040.873,-67.394,423.390,169.020,35.950,156.773
C02535=1040.867,-67.677,423.403,169.017,35.950,156.773
C02536=1040.860,-67.960,423.416,169.014,35.950,156.773
C02537=1040.853,-68.242,423.429,169.012,35.949,156.773
C02538=1040.846,-68.492,423.441,169.009,35.949,156.773
C02539=1040.841,-68.742,423.453,169.007,35.948,156.773
C02540=1040.835,-68.991,423.465,169.005,35.948,156.773
C02541=1040.828,-69.241,423.477,169.002,35.947,156.773
C02542=1040.822,-69.491,423.488,169.000,35.947,156.773
C02543=1040.817,-69.740,423.500,168.998,35.947,156.773
C02544=1040.810,-69.990,423.511,168.995,35.947,156.773
C02545=1040.804,-70.239,423.523,168.993,35.947,156.773
C02546=1040.798,-70.490,423.534,168.991,35.946,156.773
C02547=1040.792,-70.739,423.547,168.988,35.946,156.773
C02548=1040.786,-70.988,423.558,168.986,35.946,156.773
C02549=1040.780,-71.238,423.570,168.984,35.945,156.773
C02550=1040.773,-71.487,423.581,168.981,35.945,156.773
C02551=1040.768,-71.738,423.593,168.979,35.945,156.773
C02552=1040.761,-71.987,423.605,168.977,35.944,156.773
C02553=1040.755,-72.237,423.616,168.974,35.944,156.773
C02554=1040.749,-72.486,423.628,168.972,35.944,156.773
C02555=1040.743,-72.736,423.639,168.970,35.944,156.773
C02556=1040.737,-72.986,423.650,168.967,35.944,156.773
C02557=1040.731,-73.235,423.662,168.965,35.943,156.772
C02558=1040.725,-73.486,423.673,168.963,35.943,156.772
C02559=1040.719,-73.734,423.685,168.960,35.943,156.772
C02560=1040.713,-73.985,423.697,168.958,35.942,156.772
C02561=1040.707,-74.234,423.709,168.956,35.942,156.772
C02562=1040.701,-74.484,423.720,168.953,35.942,156.772
C02563=1040.694,-74.734,423.730,168.951,35.942,156.772
C02564=1040.688,-74.983,423.742,168.948,35.941,156.772
C02565=1040.682,-75.233,423.753,168.946,35.941,156.772
C02566=1040.676,-75.482,423.764,168.944,35.941,156.772
C02567=1040.669,-75.732,423.776,168.941,35.941,156.772
C02568=1040.663,-75.982,423.787,168.939,35.941,156.772
C02569=1040.657,-76.232,423.798,168.936,35.941,156.772
C02570=1040.651,-76.482,423.809,168.934,35.941,156.772
C02571=1040.645,-76.731,423.821,168.932,35.941,156.772
C02572=1040.638,-76.981,423.832,168.929,35.941,156.772
C02573=1040.633,-77.230,423.843,168.927,35.941,156.772
C02574=1040.626,-77.480,423.855,168.924,35.940,156.772
C02575=1040.620,-77.729,423.866,168.922,35.940,156.772
C02576=1040.614,-77.980,423.877,168.920,35.940,156.772
C02577=1040.608,-78.229,423.888,168.917,35.940,156.772
C02578=1040.602,-78.479,423.900,168.915,35.940,156.772
C02579=1040.596,-78.728,423.911,168.912,35.940,156.772
C02580=1040.589,-78.978,423.922,168.910,35.940,156.772
C02581=1040.584,-79.228,423.933,168.908,35.940,156.772
C02582=1040.577,-79.478,423.944,168.905,35.940,156.772
C02583=1040.571,-79.727,423.955,168.903,35.939,156.772
C02584=1040.564,-79.977,423.966,168.900,35.939,156.772
C02585=1040.559,-80.226,423.977,168.898,35.939,156.772
C02586=1040.552,-80.477,423.989,168.896,35.939,156.772
C02587=1040.546,-80.726,423.999,168.893,35.939,156.772
C02588=1040.539,-80.976,424.010,168.891,35.939,156.772
C02589=1040.534,-81.225,424.021,168.888,35.939,156.772
C02590=1040.527,-81.475,424.032,168.886,35.939,156.772
C02591=1040.521,-81.725,424.042,168.883,35.939,156.772
C02592=1040.514,-81.975,424.054,168.881,35.939,156.772
C02593=1040.508,-82.223,424.065,168.878,35.939,156.772
C02594=1040.502,-82.473,424.076,168.876,35.939,156.772
C02595=1040.496,-82.723,424.087,168.874,35.939,156.772
C02596=1040.490,-82.973,424.098,168.871,35.939,156.772
C02597=1040.483,-83.223,424.108,168.869,35.939,156.772
C02598=1040.476,-83.507,424.120,168.866,35.939,156.772
C02599=1040.469,-83.793,424.133,168.863,35.939,156.772
C02600=1040.461,-84.078,424.145,168.860,35.939,156.772
C02601=1040.454,-84.362,424.158,168.858,35.939,156.772
C02602=1040.448,-84.612,424.169,168.855,35.939,156.772
C02603=1040.442,-84.862,424.180,168.853,35.939,156.772
C02604=1040.436,-85.111,424.190,168.850,35.939,156.773
C02605=1040.429,-85.361,424.201,168.848,35.939,156.773
C02606=1040.424,-85.611,424.211,168.845,35.939,156.773
C02607=1040.417,-85.861,424.222,168.843,35.939,156.773
C02608=1040.411,-86.110,424.233,168.840,35.939,156.773
C02609=1040.405,-86.360,424.244,168.838,35.939,156.773
C02610=1040.398,-86.610,424.254,168.835,35.939,156.773
C02611=1040.393,-86.859,424.265,168.833,35.939,156.773
C02612=1040.387,-87.109,424.276,168.831,35.939,156.773
C02613=1040.380,-87.359,424.287,168.828,35.940,156.773
C02614=1040.374,-87.608,424.298,168.826,35.940,156.773
C02615=1040.368,-87.858,424.309,168.823,35.940,156.773
C02616=1040.361,-88.108,424.319,168.821,35.940,156.773
C02617=1040.356,-88.358,424.329,168.818,35.940,156.773
C02618=1040.350,-88.607,424.340,168.816,35.939,156.773
C02619=1040.343,-88.857,424.351,168.813,35.939,156.773
C02620=1040.337,-89.106,424.362,168.811,35.939,156.773
C02621=1040.331,-89.356,424.372,168.808,35.940,156.773
C02622=1040.324,-89.606,424.383,168.806,35.940,156.773
C02623=1040.319,-89.856,424.393,168.803,35.940,156.773
C02624=1040.313,-90.105,424.404,168.801,35.940,156.773
C02625=1040.307,-90.355,424.415,168.798,35.940,156.773
C02626=1040.300,-90.605,424.425,168.796,35.940,156.773
C02627=1040.294,-90.855,424.435,168.794,35.940,156.773
C02628=1040.289,-91.104,424.446,168.791,35.940,156.773
C02629=1040.282,-91.353,424.457,168.789,35.940,156.773
C02630=1040.276,-91.603,424.468,168.786,35.940,156.773
C02631=1040.270,-91.854,424.478,168.784,35.940,156.773
C02632=1040.264,-92.103,424.488,168.781,35.940,156.773
C02633=1040.258,-92.352,424.499,168.779,35.940,156.773
C02634=1040.251,-92.602,424.510,168.776,35.941,156.773
C02635=1040.246,-92.852,424.520,168.774,35.941,156.773
C02636=1040.239,-93.101,424.530,168.771,35.941,156.773
C02637=1040.233,-93.351,424.541,168.769,35.941,156.773
C02638=1040.228,-93.601,424.551,168.766,35.941,156.773
C02639=1040.221,-93.851,424.562,168.764,35.941,156.773
C02640=1040.215,-94.100,424.573,168.761,35.941,156.773
C02641=1040.209,-94.350,424.582,168.759,35.941,156.773
C02642=1040.203,-94.600,424.593,168.756,35.941,156.773
C02643=1040.197,-94.849,424.604,168.754,35.941,156.773
C02644=1040.191,-95.100,424.614,168.751,35.942,156.774
C02645=1040.185,-95.349,424.625,168.749,35.942,156.774
C02646=1040.179,-95.598,424.635,168.746,35.942,156.774
C02647=1040.173,-95.848,424.645,168.744,35.942,156.774
C02648=1040.167,-96.098,424.656,168.742,35.942,156.774
C02649=1040.161,-96.348,424.666,168.740,35.942,156.774
C02650=1040.155,-96.597,424.677,168.738,35.942,156.774
C02651=1040.148,-96.847,424.687,168.735,35.942,156.774
C02652=1040.143,-97.097,424.697,168.733,35.942,156.774
C02653=1040.136,-97.346,424.708,168.730,35.943,156.774
C02654=1040.131,-97.597,424.718,168.728,35.943,156.774
C02655=1040.125,-97.846,424.728,168.725,35.943,156.774
C02656=1040.118,-98.095,424.738,168.723,35.943,156.774
C02657=1040.113,-98.345,424.749,168.720,35.943,156.774
C02658=1040.106,-98.595,424.759,168.718,35.943,156.774
C02659=1040.099,-98.845,424.769,168.715,35.944,156.774
C02660=1040.094,-99.095,424.779,168.712,35.944,156.774
C02661=1040.088,-99.345,424.789,168.710,35.944,156.774
C02662=1040.081,-99.585,424.798,168.708,35.944,156.774
C02663=1040.076,-99.826,424.809,168.705,35.945,156.774
C02664=1040.069,-100.067,424.818,168.703,35.945,156.774
C02665=1040.064,-100.308,424.828,168.700,35.945,156.774
C02666=1040.058,-100.548,424.838,168.698,35.946,156.775
C02667=1040.053,-100.790,424.847,168.695,35.945,156.775
C02668=1040.046,-101.030,424.857,168.693,35.946,156.775
C02669=1040.041,-101.271,424.867,168.690,35.946,156.775
C02670=1040.034,-101.521,424.877,168.688,35.947,156.775
C02671=1040.028,-101.770,424.886,168.685,35.947,156.775
C02672=1040.023,-102.020,424.897,168.683,35.947,156.775
C02673=1040.016,-102.270,424.907,168.680,35.947,156.775
C02674=1040.010,-102.520,424.917,168.678,35.947,156.775
C02675=1040.003,-102.769,424.927,168.675,35.948,156.775
C02676=1039.998,-103.019,424.937,168.673,35.948,156.775
C02677=1039.991,-103.269,424.947,168.670,35.948,156.775
C02678=1039.985,-103.518,424.957,168.668,35.948,156.775
C02679=1039.979,-103.768,424.966,168.665,35.949,156.775
C02680=1039.973,-104.018,424.977,168.663,35.949,156.775
C02681=1039.967,-104.267,424.987,168.660,35.950,156.775
C02682=1039.961,-104.517,424.996,168.658,35.950,156.775
C02683=1039.955,-104.767,425.006,168.656,35.950,156.776
C02684=1039.949,-105.017,425.016,168.653,35.950,156.776
C02685=1039.943,-105.266,425.026,168.651,35.951,156.776
C02686=1039.937,-105.516,425.036,168.648,35.951,156.776
C02687=1039.930,-105.766,425.046,168.646,35.951,156.776
C02688=1039.925,-106.016,425.056,168.643,35.952,156.776
C02689=1039.919,-106.266,425.065,168.641,35.952,156.776
C02690=1039.912,-106.515,425.076,168.638,35.952,156.776
C02691=1039.906,-106.765,425.085,168.636,35.952,156.776
C02692=1039.900,-107.015,425.095,168.633,35.953,156.776
C02693=1039.894,-107.265,425.105,168.631,35.953,156.776
C02694=1039.888,-107.515,425.114,168.628,35.954,156.776
C02695=1039.882,-107.764,425.124,168.625,35.954,156.776
C02696=1039.876,-108.014,425.134,168.623,35.954,156.776
C02697=1039.869,-108.263,425.144,168.620,35.955,156.777
C02698=1039.863,-108.513,425.153,168.618,35.955,156.777
C02699=1039.857,-108.763,425.163,168.615,35.955,156.777
C02700=1039.852,-109.012,425.172,168.613,35.956,156.777
C02701=1039.845,-109.262,425.182,168.610,35.957,156.777
C02702=1039.840,-109.512,425.192,168.607,35.957,156.777
C02703=1039.834,-109.762,425.202,168.605,35.957,156.777
C02704=1039.828,-110.012,425.211,168.602,35.958,156.777
C02705=1039.821,-110.261,425.221,168.600,35.958,156.777
C02706=1039.814,-110.566,425.233,168.597,35.958,156.777
C02707=1039.806,-110.871,425.244,168.594,35.959,156.777
C02708=1039.799,-111.176,425.256,168.591,35.960,156.778
C02709=1039.792,-111.481,425.268,168.588,35.960,156.778
C02710=1039.785,-111.730,425.278,168.586,35.960,156.778
C02711=1039.779,-111.980,425.287,168.583,35.961,156.778
C02712=1039.773,-112.231,425.296,168.580,35.961,156.778
C02713=1039.767,-112.480,425.306,168.578,35.962,156.778
C02714=1039.761,-112.730,425.315,168.575,35.962,156.778
C02715=1039.755,-112.980,425.325,168.573,35.963,156.778
C02716=1039.749,-113.229,425.334,168.570,35.963,156.778
C02717=1039.743,-113.479,425.343,168.568,35.963,156.778
C02718=1039.737,-113.729,425.353,168.565,35.964,156.778
C02719=1039.731,-113.978,425.363,168.562,35.964,156.779
C02720=1039.725,-114.228,425.372,168.560,35.965,156.779
C02721=1039.718,-114.478,425.382,168.557,35.965,156.779
C02722=1039.712,-114.728,425.391,168.555,35.966,156.779
C02723=1039.707,-114.977,425.400,168.552,35.966,156.779
C02724=1039.701,-115.227,425.410,168.549,35.967,156.779
C02725=1039.695,-115.477,425.419,168.547,35.967,156.779
C02726=1039.688,-115.763,425.430,168.544,35.968,156.779
C02727=1039.680,-116.049,425.441,168.542,35.969,156.779
C02728=1039.673,-116.336,425.452,168.539,35.969,156.780
C02729=1039.667,-116.623,425.462,168.536,35.970,156.780
C02730=1039.660,-116.871,425.471,168.533,35.970,156.780
C02731=1039.654,-117.121,425.481,168.531,35.971,156.780
C02732=1039.648,-117.372,425.489,168.528,35.971,156.780
C02733=1039.642,-117.621,425.499,168.526,35.972,156.780
C02734=1039.637,-117.871,425.508,168.523,35.972,156.780
C02735=1039.631,-118.120,425.518,168.520,35.973,156.780
C02736=1039.625,-118.371,425.527,168.518,35.974,156.780
C02737=1039.618,-118.621,425.536,168.515,35.974,156.781
C02738=1039.612,-118.870,425.546,168.513,35.975,156.781
C02739=1039.606,-119.119,425.554,168.510,35.975,156.781
C02740=1039.600,-119.370,425.563,168.507,35.975,156.781
C02741=1039.594,-119.619,425.573,168.505,35.976,156.781
C02742=1039.588,-119.869,425.582,168.502,35.977,156.781
C02743=1039.583,-120.119,425.591,168.500,35.977,156.781
C02744=1039.576,-120.369,425.600,168.497,35.978,156.781
C02745=1039.569,-120.618,425.609,168.495,35.979,156.781
C02746=1039.564,-120.868,425.618,168.493,35.979,156.781
C02747=1039.558,-121.118,425.627,168.490,35.980,156.782
C02748=1039.552,-121.367,425.637,168.487,35.980,156.782
C02749=1039.546,-121.618,425.646,168.485,35.981,156.782
C02750=1039.540,-121.867,425.655,168.482,35.982,156.782
C02751=1039.533,-122.116,425.664,168.480,35.982,156.782
C02752=1039.528,-122.367,425.673,168.477,35.983,156.782
C02753=1039.522,-122.616,425.682,168.474,35.983,156.782
C02754=1039.516,-122.866,425.691,168.472,35.984,156.782
C02755=1039.510,-123.116,425.701,168.469,35.985,156.783
C02756=1039.504,-123.365,425.709,168.467,35.985,156.783
C02757=1039.498,-123.615,425.718,168.464,35.986,156.783
C02758=1039.492,-123.865,425.728,168.461,35.987,156.783
C02759=1039.486,-124.115,425.736,168.459,35.987,156.783
C02760=1039.479,-124.364,425.745,168.456,35.988,156.783
C02761=1039.474,-124.615,425.754,168.454,35.988,156.783
C02762=1039.468,-124.864,425.763,168.452,35.989,156.783
C02763=1039.461,-125.114,425.771,168.449,35.990,156.784
C02764=1039.455,-125.364,425.781,168.447,35.990,156.784
C02765=1039.450,-125.614,425.789,168.444,35.991,156.784
C02766=1039.443,-125.863,425.798,168.441,35.992,156.784
C02767=1039.437,-126.113,425.807,168.439,35.993,156.784
C02768=1039.432,-126.363,425.816,168.436,35.993,156.784
C02769=1039.425,-126.613,425.825,168.433,35.994,156.784
C02770=1039.419,-126.862,425.834,168.431,35.995,156.784
C02771=1039.414,-127.112,425.843,168.428,35.995,156.785
C02772=1039.407,-127.362,425.851,168.425,35.996,156.785
C02773=1039.401,-127.611,425.860,168.423,35.997,156.785
C02774=1039.396,-127.862,425.869,168.420,35.998,156.785
C02775=1039.390,-128.111,425.878,168.418,35.998,156.785
C02776=1039.386,-128.361,425.889,168.415,35.998,156.785
C02777=1039.382,-128.610,425.899,168.413,35.997,156.785
C02778=1039.379,-128.861,425.911,168.411,35.996,156.785
C02779=1039.377,-129.110,425.922,168.409,35.994,156.785
C02780=1039.376,-129.360,425.935,168.407,35.992,156.784
C02781=1039.376,-129.610,425.947,168.406,35.990,156.784
C02782=1039.376,-129.860,425.961,168.404,35.987,156.783
C02783=1039.378,-130.110,425.976,168.402,35.983,156.783
C02784=1039.379,-130.361,425.990,168.401,35.980,156.782
C02785=1039.382,-130.610,426.005,168.400,35.975,156.781
C02786=1039.385,-130.861,426.021,168.398,35.971,156.781
C02787=1039.390,-131.111,426.038,168.397,35.965,156.780
C02788=1039.395,-131.361,426.055,168.396,35.959,156.779
C02789=1039.401,-131.611,426.073,168.395,35.954,156.778
C02790=1039.057,-131.635,425.810,168.347,36.153,156.812
C02791=1039.051,-131.385,425.792,168.348,36.160,156.813
C02792=1039.046,-131.135,425.775,168.349,36.165,156.814
C02793=1039.042,-130.885,425.758,168.351,36.170,156.814
C02794=1039.038,-130.634,425.741,168.352,36.176,156.815
C02795=1039.035,-130.384,425.726,168.354,36.180,156.816
C02796=1039.033,-130.134,425.712,168.355,36.183,156.817
C02797=1039.032,-129.885,425.698,168.356,36.187,156.817
C02798=1039.032,-129.635,425.684,168.358,36.189,156.818
C02799=1039.032,-129.384,425.671,168.360,36.192,156.818
C02800=1039.033,-129.135,425.659,168.362,36.194,156.818
C02801=1039.035,-128.884,425.646,168.364,36.196,156.819
C02802=1039.038,-128.635,425.636,168.366,36.197,156.819
C02803=1039.041,-128.385,425.625,168.368,36.197,156.819
C02804=1039.046,-128.135,425.615,168.370,36.198,156.819
C02805=1039.052,-127.885,425.605,168.373,36.197,156.819
C02806=1039.057,-127.636,425.596,168.375,36.197,156.819
C02807=1039.063,-127.387,425.588,168.378,36.196,156.819
C02808=1039.069,-127.136,425.579,168.381,36.196,156.819
C02809=1039.075,-126.886,425.570,168.383,36.195,156.819
C02810=1039.081,-126.637,425.561,168.386,36.194,156.818
C02811=1039.087,-126.387,425.553,168.389,36.193,156.818
C02812=1039.093,-126.138,425.543,168.391,36.192,156.818
C02813=1039.099,-125.888,425.535,168.394,36.192,156.818
C02814=1039.105,-125.638,425.526,168.397,36.191,156.818
C02815=1039.111,-125.388,425.517,168.399,36.190,156.818
C02816=1039.118,-125.139,425.508,168.402,36.189,156.817
C02817=1039.123,-124.888,425.499,168.404,36.188,156.817
C02818=1039.129,-124.639,425.490,168.406,36.188,156.817
C02819=1039.136,-124.389,425.482,168.409,36.187,156.817
C02820=1039.142,-124.139,425.472,168.412,36.187,156.817
C02821=1039.147,-123.889,425.464,168.414,36.186,156.817
C02822=1039.153,-123.640,425.454,168.417,36.185,156.817
C02823=1039.160,-123.390,425.446,168.419,36.185,156.817
C02824=1039.165,-123.141,425.437,168.422,36.184,156.817
C02825=1039.171,-122.890,425.428,168.425,36.183,156.816
C02826=1039.177,-122.640,425.418,168.427,36.183,156.816
C02827=1039.183,-122.391,425.409,168.430,36.182,156.816
C02828=1039.190,-122.141,425.401,168.433,36.181,156.816
C02829=1039.196,-121.891,425.391,168.435,36.181,156.816
C02830=1039.201,-121.642,425.383,168.438,36.180,156.816
C02831=1039.207,-121.392,425.373,168.440,36.180,156.816
C02832=1039.213,-121.142,425.364,168.443,36.179,156.816
C02833=1039.220,-120.892,425.355,168.445,36.178,156.815
C02834=1039.226,-120.643,425.346,168.447,36.178,156.815
C02835=1039.232,-120.393,425.337,168.450,36.177,156.815
C02836=1039.238,-120.143,425.328,168.453,36.176,156.815
C02837=1039.243,-119.893,425.319,168.455,36.176,156.815
C02838=1039.249,-119.644,425.309,168.458,36.175,156.815
C02839=1039.256,-119.394,425.301,168.460,36.175,156.815
C02840=1039.262,-119.144,425.291,168.463,36.174,156.815
C02841=1039.268,-118.895,425.282,168.466,36.173,156.815
C02842=1039.274,-118.645,425.272,168.468,36.173,156.814
C02843=1039.280,-118.394,425.264,168.471,36.172,156.814
C02844=1039.286,-118.145,425.254,168.474,36.171,156.814
C02845=1039.291,-117.896,425.245,168.476,36.171,156.814
C02846=1039.298,-117.646,425.236,168.479,36.170,156.814
C02847=1039.304,-117.396,425.227,168.481,36.169,156.814
C02848=1039.310,-117.146,425.217,168.484,36.169,156.814
C02849=1039.317,-116.896,425.208,168.486,36.168,156.814
C02850=1039.322,-116.647,425.199,168.488,36.168,156.814
C02851=1039.329,-116.360,425.188,168.491,36.167,156.813
C02852=1039.336,-116.074,425.177,168.494,36.166,156.813
C02853=1039.343,-115.787,425.167,168.497,36.166,156.813
C02854=1039.350,-115.501,425.156,168.500,36.165,156.813
C02855=1039.356,-115.251,425.146,168.503,36.165,156.813
C02856=1039.362,-115.002,425.138,168.505,36.164,156.813
C02857=1039.368,-114.752,425.128,168.508,36.164,156.813
C02858=1039.375,-114.503,425.118,168.511,36.163,156.813
C02859=1039.381,-114.253,425.109,168.513,36.163,156.813
C02860=1039.387,-114.002,425.100,168.516,36.162,156.812
C02861=1039.393,-113.753,425.090,168.519,36.162,156.812
C02862=1039.399,-113.503,425.081,168.521,36.161,156.812
C02863=1039.405,-113.254,425.072,168.524,36.161,156.812
C02864=1039.411,-113.004,425.062,168.526,36.160,156.812
C02865=1039.416,-112.754,425.052,168.529,36.159,156.812
C02866=1039.422,-112.504,425.042,168.531,36.159,156.812
C02867=1039.428,-112.254,425.033,168.533,36.159,156.812
C02868=1039.435,-112.004,425.023,168.536,36.158,156.812
C02869=1039.441,-111.755,425.014,168.538,36.158,156.812
C02870=1039.446,-111.506,425.004,168.541,36.158,156.812
C02871=1039.453,-111.256,424.995,168.543,36.157,156.811
C02872=1039.459,-111.006,424.985,168.546,36.156,156.811
C02873=1039.465,-110.756,424.976,168.549,36.156,156.811
C02874=1039.471,-110.506,424.966,168.551,36.156,156.811
C02875=1039.477,-110.257,424.957,168.554,36.155,156.811
C02876=1039.483,-110.007,424.947,168.556,36.154,156.811
C02877=1039.490,-109.757,424.937,168.559,36.154,156.811
C02878=1039.496,-109.507,424.928,168.562,36.154,156.811
C02879=1039.502,-109.257,424.918,168.564,36.153,156.811
C02880=1039.508,-109.008,424.909,168.567,36.153,156.811
C02881=1039.514,-108.757,424.899,168.569,36.153,156.811
C02882=1039.520,-108.508,424.889,168.572,36.152,156.811
C02883=1039.526,-108.259,424.879,168.574,36.151,156.810
C02884=1039.532,-108.009,424.870,168.577,36.151,156.810
C02885=1039.538,-107.760,424.860,168.580,36.151,156.810
C02886=1039.544,-107.510,424.850,168.582,36.150,156.810
C02887=1039.550,-107.260,424.841,168.585,36.150,156.810
C02888=1039.556,-107.010,424.831,168.587,36.149,156.810
C02889=1039.562,-106.760,424.821,168.589,36.149,156.810
C02890=1039.568,-106.511,424.811,168.591,36.149,156.810
C02891=1039.575,-106.261,424.801,168.594,36.148,156.810
C02892=1039.581,-106.011,424.792,168.597,36.148,156.810
C02893=1039.587,-105.762,424.782,168.599,36.148,156.810
C02894=1039.592,-105.511,424.772,168.602,36.147,156.810
C02895=1039.599,-105.262,424.762,168.604,36.147,156.810
C02896=1039.605,-105.012,424.752,168.607,36.146,156.809
C02897=1039.611,-104.763,424.743,168.609,36.146,156.809
C02898=1039.617,-104.513,424.732,168.612,36.146,156.809
C02899=1039.623,-104.263,424.722,168.615,36.146,156.809
C02900=1039.629,-104.014,424.713,168.617,36.145,156.809
C02901=1039.635,-103.764,424.703,168.620,36.145,156.809
C02902=1039.641,-103.514,424.693,168.622,36.145,156.809
C02903=1039.647,-103.264,424.683,168.625,36.144,156.809
C02904=1039.653,-103.015,424.673,168.627,36.144,156.809
C02905=1039.660,-102.765,424.663,168.630,36.143,156.809
C02906=1039.665,-102.515,424.653,168.632,36.143,156.809
C02907=1039.672,-102.265,424.643,168.635,36.143,156.809
C02908=1039.678,-102.015,424.633,168.637,36.143,156.809
C02909=1039.684,-101.766,424.622,168.640,36.142,156.809
C02910=1039.690,-101.516,424.613,168.643,36.142,156.809
C02911=1039.696,-101.266,424.603,168.645,36.142,156.808
C02912=1039.702,-101.017,424.592,168.648,36.142,156.808
C02913=1039.708,-100.767,424.583,168.650,36.141,156.808
C02914=1039.714,-100.517,424.573,168.653,36.141,156.808
C02915=1039.722,-100.230,424.561,168.656,36.140,156.808
C02916=1039.729,-99.943,424.549,168.658,36.140,156.808
C02917=1039.736,-99.655,424.538,168.660,36.140,156.808
C02918=1039.743,-99.368,424.525,168.663,36.140,156.808
C02919=1039.749,-99.118,424.516,168.666,36.139,156.808
C02920=1039.755,-98.869,424.506,168.668,36.139,156.808
C02921=1039.762,-98.619,424.496,168.671,36.139,156.808
C02922=1039.767,-98.369,424.486,168.674,36.139,156.808
C02923=1039.774,-98.120,424.476,168.676,36.138,156.808
C02924=1039.780,-97.870,424.466,168.679,36.138,156.808
C02925=1039.786,-97.620,424.455,168.681,36.137,156.808
C02926=1039.792,-97.370,424.445,168.684,36.137,156.808
C02927=1039.798,-97.121,424.434,168.686,36.137,156.808
C02928=1039.804,-96.871,424.425,168.689,36.137,156.807
C02929=1039.810,-96.622,424.414,168.691,36.137,156.807
C02930=1039.816,-96.372,424.404,168.694,36.137,156.807
C02931=1039.822,-96.122,424.393,168.696,36.137,156.807
C02932=1039.828,-95.873,424.383,168.699,36.136,156.807
C02933=1039.834,-95.622,424.373,168.701,36.136,156.807
C02934=1039.840,-95.373,424.362,168.704,36.136,156.807
C02935=1039.847,-95.124,424.351,168.706,36.136,156.807
C02936=1039.852,-94.874,424.341,168.709,36.136,156.807
C02937=1039.858,-94.624,424.331,168.711,36.136,156.807
C02938=1039.864,-94.374,424.321,168.714,36.136,156.807
C02939=1039.870,-94.124,424.310,168.716,36.136,156.807
C02940=1039.877,-93.875,424.299,168.719,36.135,156.807
C02941=1039.882,-93.625,424.289,168.721,36.135,156.807
C02942=1039.889,-93.376,424.279,168.724,36.135,156.807
C02943=1039.899,-92.954,424.261,168.728,36.135,156.807
C02944=1039.909,-92.532,424.242,168.732,36.135,156.807
C02945=1039.919,-92.110,424.225,168.736,36.135,156.807
C02946=1039.930,-91.688,424.207,168.740,36.134,156.807
C02947=1039.936,-91.439,424.197,168.743,36.134,156.807
C02948=1039.942,-91.189,424.187,168.745,36.134,156.807
C02949=1039.947,-90.939,424.176,168.748,36.134,156.807
C02950=1039.955,-90.689,424.165,168.750,36.134,156.807
C02951=1039.960,-90.440,424.154,168.753,36.133,156.807
C02952=1039.966,-90.190,424.144,168.755,36.134,156.807
C02953=1039.972,-89.941,424.134,168.758,36.134,156.807
C02954=1039.979,-89.690,424.123,168.760,36.134,156.807
C02955=1039.985,-89.441,424.112,168.763,36.134,156.807
C02956=1039.991,-89.192,424.102,168.765,36.133,156.806
C02957=1039.997,-88.942,424.090,168.768,36.133,156.806
C02958=1040.003,-88.692,424.081,168.770,36.133,156.806
C02959=1040.009,-88.442,424.070,168.773,36.133,156.806
C02960=1040.015,-88.193,424.059,168.775,36.133,156.806
C02961=1040.022,-87.943,424.048,168.778,36.133,156.806
C02962=1040.028,-87.693,424.038,168.779,36.132,156.806
C02963=1040.034,-87.444,424.027,168.782,36.132,156.806
C02964=1040.040,-87.194,424.016,168.784,36.132,156.806
C02965=1040.046,-86.944,424.006,168.787,36.133,156.806
C02966=1040.052,-86.695,423.996,168.789,36.133,156.806
C02967=1040.059,-86.445,423.984,168.792,36.133,156.806
C02968=1040.064,-86.195,423.973,168.794,36.132,156.806
C02969=1040.071,-85.945,423.963,168.796,36.132,156.806
C02970=1040.077,-85.696,423.952,168.799,36.132,156.806
C02971=1040.083,-85.446,423.941,168.801,36.132,156.806
C02972=1040.090,-85.196,423.930,168.804,36.132,156.806
C02973=1040.096,-84.947,423.920,168.806,36.132,156.806
C02974=1040.101,-84.697,423.909,168.809,36.132,156.806
C02975=1040.111,-84.334,423.893,168.812,36.131,156.806
C02976=1040.120,-83.972,423.877,168.816,36.132,156.806
C02977=1040.129,-83.609,423.862,168.820,36.132,156.806
C02978=1040.139,-83.247,423.846,168.823,36.132,156.806
C02979=1040.144,-82.997,423.835,168.826,36.132,156.806
C02980=1040.150,-82.748,423.824,168.828,36.132,156.806
C02981=1040.157,-82.498,423.813,168.831,36.132,156.806
C02982=1040.163,-82.248,423.802,168.833,36.131,156.806
C02983=1040.169,-81.998,423.791,168.835,36.131,156.806
C02984=1040.176,-81.749,423.781,168.838,36.131,156.806
C02985=1040.182,-81.499,423.770,168.840,36.131,156.806
C02986=1040.188,-81.249,423.759,168.843,36.131,156.806
C02987=1040.195,-80.999,423.748,168.845,36.131,156.806
C02988=1040.201,-80.750,423.737,168.848,36.131,156.806
C02989=1040.207,-80.500,423.725,168.850,36.131,156.806
C02990=1040.214,-80.251,423.715,168.853,36.131,156.806
C02991=1040.220,-80.001,423.704,168.855,36.131,156.806
C02992=1040.226,-79.751,423.693,168.858,36.131,156.806
C02993=1040.232,-79.501,423.682,168.860,36.131,156.806
C02994=1040.238,-79.252,423.671,168.862,36.131,156.806
C02995=1040.245,-79.002,423.659,168.865,36.131,156.806
C02996=1040.250,-78.753,423.648,168.867,36.131,156.806
C02997=1040.257,-78.502,423.637,168.870,36.131,156.806
C02998=1040.262,-78.253,423.626,168.872,36.131,156.806
C02999=1040.269,-78.003,423.615,168.874,36.131,156.806
C03000=1040.276,-77.754,423.604,168.877,36.131,156.806
C03001=1040.282,-77.504,423.592,168.879,36.131,156.806
C03002=1040.288,-77.254,423.582,168.882,36.132,156.806
C03003=1040.294,-77.004,423.570,168.884,36.132,156.806
C03004=1040.300,-76.755,423.559,168.887,36.132,156.806
C03005=1040.306,-76.505,423.547,168.889,36.132,156.806
C03006=1040.312,-76.256,423.537,168.891,36.132,156.806
C03007=1040.319,-76.006,423.525,168.894,36.132,156.806
C03008=1040.324,-75.757,423.514,168.896,36.132,156.806
C03009=1040.331,-75.506,423.502,168.899,36.132,156.806
C03010=1040.337,-75.258,423.491,168.901,36.132,156.806
C03011=1040.343,-75.007,423.480,168.903,36.133,156.806
C03012=1040.349,-74.758,423.469,168.906,36.133,156.806
C03013=1040.356,-74.508,423.457,168.908,36.133,156.806
C03014=1040.362,-74.258,423.446,168.911,36.133,156.806
C03015=1040.368,-74.009,423.435,168.913,36.133,156.806
C03016=1040.374,-73.759,423.423,168.915,36.133,156.806
C03017=1040.380,-73.510,423.412,168.918,36.134,156.806
C03018=1040.386,-73.259,423.401,168.920,36.134,156.806
C03019=1040.392,-73.010,423.388,168.922,36.134,156.806
C03020=1040.398,-72.760,423.377,168.925,36.135,156.806
C03021=1040.405,-72.510,423.365,168.927,36.135,156.806
C03022=1040.410,-72.261,423.354,168.929,36.135,156.806
C03023=1040.417,-72.011,423.342,168.932,36.135,156.806
C03024=1040.422,-71.762,423.331,168.934,36.135,156.806
C03025=1040.429,-71.512,423.319,168.937,36.135,156.806
C03026=1040.434,-71.263,423.308,168.939,36.136,156.806
C03027=1040.441,-71.013,423.296,168.941,36.136,156.806
C03028=1040.447,-70.762,423.284,168.944,36.136,156.806
C03029=1040.453,-70.514,423.273,168.946,36.137,156.806
C03030=1040.459,-70.263,423.261,168.948,36.137,156.806
C03031=1040.465,-70.015,423.250,168.951,36.137,156.806
C03032=1040.471,-69.765,423.237,168.954,36.137,156.806
C03033=1040.477,-69.514,423.226,168.956,36.137,156.806
C03034=1040.483,-69.266,423.214,168.959,36.137,156.806
C03035=1040.490,-69.015,423.203,168.961,36.138,156.807
C03036=1040.495,-68.766,423.191,168.963,36.138,156.807
C03037=1040.501,-68.516,423.180,168.966,36.139,156.807
C03038=1040.508,-68.266,423.168,168.968,36.139,156.807
C03039=1040.515,-67.984,423.155,168.971,36.139,156.807
C03040=1040.522,-67.701,423.142,168.973,36.140,156.807
C03041=1040.529,-67.418,423.128,168.976,36.140,156.807
C03042=1040.536,-67.136,423.115,168.979,36.140,156.807
C03043=1040.543,-66.886,423.103,168.981,36.140,156.807
C03044=1040.548,-66.636,423.091,168.983,36.140,156.807
C03045=1040.554,-66.387,423.079,168.986,36.141,156.807
C03046=1040.561,-66.137,423.067,168.988,36.141,156.807
C03047=1040.566,-65.887,423.056,168.990,36.141,156.807
C03048=1040.573,-65.638,423.044,168.993,36.142,156.807
C03049=1040.579,-65.388,423.032,168.995,36.142,156.807
C03050=1040.585,-65.139,423.021,168.997,36.142,156.807
C03051=1040.591,-64.889,423.009,169.000,36.142,156.807
C03052=1040.597,-64.639,422.997,169.002,36.142,156.807
C03053=1040.604,-64.390,422.985,169.004,36.143,156.807
C03054=1040.609,-64.140,422.973,169.007,36.143,156.807
C03055=1040.616,-63.890,422.961,169.009,36.144,156.807
C03056=1040.622,-63.641,422.949,169.011,36.144,156.807
C03057=1040.629,-63.391,422.937,169.014,36.144,156.807
C03058=1040.634,-63.141,422.926,169.016,36.144,156.807
C03059=1040.641,-62.892,422.914,169.018,36.144,156.807
C03060=1040.647,-62.642,422.902,169.021,36.145,156.808
C03061=1040.653,-62.392,422.889,169.023,36.145,156.808
C03062=1040.659,-62.143,422.878,169.025,36.145,156.808
C03063=1040.666,-61.893,422.867,169.028,36.146,156.808
C03064=1040.672,-61.643,422.854,169.030,36.146,156.808
C03065=1040.678,-61.394,422.842,169.032,36.147,156.808
C03066=1040.685,-61.144,422.830,169.035,36.147,156.808
C03067=1040.691,-60.895,422.818,169.037,36.147,156.808
C03068=1040.697,-60.646,422.806,169.039,36.147,156.808
C03069=1040.703,-60.395,422.795,169.042,36.147,156.808
C03070=1040.710,-60.146,422.783,169.044,36.148,156.808
C03071=1040.716,-59.896,422.770,169.046,36.148,156.808
C03072=1040.722,-59.646,422.758,169.049,36.149,156.808
C03073=1040.728,-59.397,422.747,169.051,36.149,156.808
C03074=1040.734,-59.148,422.734,169.053,36.149,156.808
C03075=1040.741,-58.898,422.722,169.055,36.149,156.808
C03076=1040.748,-58.648,422.710,169.058,36.150,156.808
C03077=1040.753,-58.399,422.698,169.060,36.150,156.808
C03078=1040.760,-58.149,422.686,169.062,36.150,156.808
C03079=1040.767,-57.899,422.674,169.066,36.151,156.808
C03080=1040.773,-57.649,422.661,169.068,36.151,156.808
C03081=1040.778,-57.400,422.650,169.070,36.151,156.808
C03082=1040.785,-57.150,422.638,169.073,36.151,156.808
C03083=1040.791,-56.901,422.626,169.075,36.152,156.809
C03084=1040.798,-56.651,422.614,169.077,36.152,156.809
C03085=1040.804,-56.401,422.601,169.080,36.153,156.809
C03086=1040.810,-56.152,422.589,169.082,36.153,156.809
C03087=1040.817,-55.902,422.577,169.084,36.153,156.809
C03088=1040.823,-55.652,422.565,169.086,36.154,156.809
C03089=1040.830,-55.403,422.552,169.089,36.154,156.809
C03090=1040.836,-55.154,422.540,169.091,36.154,156.809
C03091=1040.842,-54.904,422.528,169.093,36.154,156.809
C03092=1040.849,-54.654,422.516,169.096,36.155,156.809
C03093=1040.856,-54.405,422.504,169.098,36.155,156.809
C03094=1040.861,-54.155,422.491,169.100,36.156,156.809
C03095=1040.868,-53.906,422.479,169.103,36.156,156.809
C03096=1040.873,-53.656,422.467,169.105,36.156,156.809
C03097=1040.880,-53.406,422.455,169.107,36.156,156.809
C03098=1040.887,-53.157,422.443,169.109,36.157,156.809
C03099=1040.893,-52.907,422.430,169.112,36.157,156.809
C03100=1040.899,-52.657,422.418,169.114,36.158,156.809
C03101=1040.906,-52.408,422.406,169.116,36.158,156.809
C03102=1040.912,-52.158,422.393,169.119,36.158,156.810
C03103=1040.919,-51.876,422.380,169.121,36.158,156.810
C03104=1040.927,-51.595,422.366,169.124,36.159,156.810
C03105=1040.934,-51.313,422.352,169.126,36.159,156.810
C03106=1040.942,-51.032,422.338,169.129,36.160,156.810
C03107=1040.948,-50.782,422.326,169.131,36.160,156.810
C03108=1040.954,-50.532,422.313,169.133,36.160,156.810
C03109=1040.960,-50.282,422.300,169.136,36.161,156.810
C03110=1040.967,-50.034,422.288,169.138,36.161,156.810
C03111=1040.973,-49.784,422.275,169.140,36.162,156.810
C03112=1040.979,-49.534,422.263,169.142,36.162,156.810
C03113=1040.986,-49.285,422.250,169.146,36.163,156.810
C03114=1040.992,-49.035,422.237,169.148,36.163,156.810
C03115=1040.998,-48.785,422.225,169.150,36.164,156.810
C03116=1041.004,-48.535,422.212,169.152,36.164,156.810
C03117=1041.011,-48.286,422.200,169.154,36.165,156.811
C03118=1041.016,-48.036,422.187,169.157,36.165,156.811
C03119=1041.022,-47.786,422.175,169.159,36.166,156.811
C03120=1041.029,-47.537,422.161,169.161,36.166,156.811
C03121=1041.035,-47.288,422.149,169.163,36.167,156.811
C03122=1041.041,-47.038,422.136,169.166,36.167,156.811
C03123=1041.047,-46.788,422.124,169.168,36.168,156.811
C03124=1041.053,-46.539,422.111,169.170,36.168,156.811
C03125=1041.060,-46.290,422.098,169.172,36.169,156.811
C03126=1041.066,-46.040,422.086,169.174,36.169,156.811
C03127=1041.072,-45.790,422.072,169.177,36.170,156.811
C03128=1041.078,-45.541,422.060,169.179,36.170,156.811
C03129=1041.085,-45.291,422.048,169.181,36.171,156.812
C03130=1041.091,-45.042,422.035,169.183,36.171,156.812
C03131=1041.097,-44.792,422.022,169.185,36.172,156.812
C03132=1041.103,-44.543,422.009,169.188,36.172,156.812
C03133=1041.109,-44.293,421.996,169.190,36.173,156.812
C03134=1041.117,-44.043,421.983,169.192,36.173,156.812
C03135=1041.123,-43.793,421.971,169.194,36.174,156.812
C03136=1041.129,-43.544,421.957,169.197,36.174,156.812
C03137=1041.135,-43.294,421.945,169.200,36.175,156.812
C03138=1041.142,-43.045,421.932,169.202,36.175,156.812
C03139=1041.148,-42.795,421.920,169.204,36.176,156.812
C03140=1041.154,-42.546,421.906,169.206,36.176,156.812
C03141=1041.160,-42.296,421.894,169.209,36.177,156.813
C03142=1041.167,-42.046,421.880,169.211,36.178,156.813
C03143=1041.173,-41.797,421.868,169.213,36.178,156.813
C03144=1041.179,-41.547,421.855,169.215,36.178,156.813
C03145=1041.185,-41.297,421.842,169.217,36.179,156.813
C03146=1041.191,-41.048,421.829,169.219,36.180,156.813
C03147=1041.198,-40.799,421.816,169.222,36.180,156.813
C03148=1041.204,-40.549,421.804,169.224,36.180,156.813
C03149=1041.211,-40.299,421.790,169.226,36.181,156.813
C03150=1041.217,-40.049,421.778,169.228,36.182,156.813
C03151=1041.223,-39.800,421.764,169.230,36.182,156.813
C03152=1041.229,-39.551,421.751,169.233,36.182,156.813
C03153=1041.236,-39.301,421.739,169.235,36.183,156.813
C03154=1041.243,-39.051,421.726,169.237,36.184,156.814
C03155=1041.249,-38.801,421.713,169.239,36.184,156.814
C03156=1041.255,-38.552,421.700,169.241,36.185,156.814
C03157=1041.261,-38.303,421.687,169.245,36.186,156.814
C03158=1041.267,-38.053,421.674,169.247,36.186,156.814
C03159=1041.274,-37.803,421.660,169.249,36.187,156.814
C03160=1041.280,-37.554,421.647,169.251,36.188,156.814
C03161=1041.286,-37.305,421.634,169.253,36.188,156.814
C03162=1041.292,-37.055,421.621,169.255,36.188,156.814
C03163=1041.299,-36.805,421.608,169.257,36.189,156.814
C03164=1041.305,-36.555,421.594,169.260,36.190,156.815
C03165=1041.312,-36.306,421.581,169.262,36.190,156.815
C03166=1041.318,-36.056,421.569,169.264,36.191,156.815
C03167=1041.324,-35.775,421.553,169.266,36.192,156.815
C03168=1041.331,-35.495,421.539,169.269,36.192,156.815
C03169=1041.338,-35.213,421.523,169.271,36.193,156.815
C03170=1041.345,-34.932,421.509,169.273,36.194,156.815
C03171=1041.352,-34.683,421.495,169.276,36.195,156.815
C03172=1041.358,-34.433,421.482,169.278,36.195,156.815
C03173=1041.365,-34.183,421.468,169.280,36.196,156.816
C03174=1041.371,-33.934,421.455,169.282,36.196,156.816
C03175=1041.377,-33.684,421.443,169.285,36.197,156.816
C03176=1041.383,-33.435,421.429,169.287,36.198,156.816
C03177=1041.390,-33.185,421.416,169.289,36.198,156.816
C03178=1041.395,-32.936,421.402,169.292,36.199,156.816
C03179=1041.402,-32.686,421.389,169.294,36.200,156.816
C03180=1041.408,-32.436,421.375,169.296,36.200,156.816
C03181=1041.415,-32.187,421.362,169.298,36.201,156.816
C03182=1041.421,-31.938,421.348,169.300,36.202,156.817
C03183=1041.427,-31.689,421.335,169.302,36.202,156.817
C03184=1041.434,-31.438,421.322,169.304,36.203,156.817
C03185=1041.440,-31.189,421.309,169.306,36.204,156.817
C03186=1041.446,-30.939,421.296,169.309,36.204,156.817
C03187=1041.453,-30.689,421.282,169.311,36.205,156.817
C03188=1041.459,-30.440,421.269,169.313,36.206,156.817
C03189=1041.464,-30.191,421.255,169.315,36.206,156.817
C03190=1041.471,-29.941,421.241,169.317,36.207,156.817
C03191=1041.477,-29.691,421.228,169.319,36.208,156.818
C03192=1041.484,-29.442,421.215,169.322,36.208,156.818
C03193=1041.491,-29.192,421.201,169.324,36.209,156.818
C03194=1041.497,-28.943,421.188,169.327,36.210,156.818
C03195=1041.504,-28.693,421.174,169.329,36.210,156.818
C03196=1041.510,-28.444,421.161,169.331,36.211,156.818
C03197=1041.516,-28.194,421.148,169.333,36.212,156.818
C03198=1041.523,-27.944,421.134,169.335,36.212,156.818
C03199=1041.528,-27.695,421.120,169.337,36.213,156.818
C03200=1041.535,-27.445,421.106,169.339,36.213,156.819
C03201=1041.541,-27.196,421.093,169.341,36.214,156.819
C03202=1041.548,-26.946,421.080,169.343,36.215,156.819
C03203=1041.555,-26.697,421.066,169.346,36.215,156.819
C03204=1041.560,-26.447,421.052,169.348,36.216,156.819
C03205=1041.566,-26.198,421.038,169.350,36.217,156.819
C03206=1041.573,-25.948,421.025,169.352,36.217,156.819
C03207=1041.579,-25.699,421.011,169.354,36.218,156.819
C03208=1041.585,-25.449,420.997,169.357,36.219,156.820
C03209=1041.592,-25.199,420.984,169.359,36.220,156.820
C03210=1041.597,-24.950,420.969,169.361,36.221,156.820
C03211=1041.604,-24.700,420.956,169.363,36.221,156.820
C03212=1041.610,-24.451,420.942,169.365,36.222,156.820
C03213=1041.617,-24.201,420.928,169.367,36.223,156.820
C03214=1041.623,-23.952,420.915,169.369,36.224,156.820
C03215=1041.629,-23.703,420.900,169.371,36.225,156.820
C03216=1041.635,-23.453,420.887,169.373,36.225,156.821
C03217=1041.642,-23.203,420.874,169.375,36.226,156.821
C03218=1041.648,-22.953,420.859,169.378,36.227,156.821
C03219=1041.654,-22.704,420.846,169.380,36.227,156.821
C03220=1041.660,-22.454,420.831,169.382,36.228,156.821
C03221=1041.666,-22.205,420.818,169.384,36.229,156.821
C03222=1041.673,-21.955,420.804,169.387,36.230,156.821
C03223=1041.679,-21.706,420.790,169.389,36.230,156.821
C03224=1041.685,-21.457,420.776,169.391,36.231,156.822
C03225=1041.692,-21.207,420.763,169.393,36.232,156.822
C03226=1041.698,-20.957,420.749,169.395,36.232,156.822
C03227=1041.705,-20.708,420.734,169.397,36.233,156.822
C03228=1041.710,-20.458,420.721,169.399,36.234,156.822
C03229=1041.717,-20.208,420.707,169.401,36.235,156.822
C03230=1041.723,-19.960,420.693,169.403,36.236,156.822
C03231=1041.731,-19.677,420.678,169.406,36.236,156.822
C03232=1041.738,-19.396,420.662,169.408,36.238,156.823
C03233=1041.744,-19.114,420.645,169.410,36.238,156.823
C03234=1041.752,-18.832,420.630,169.412,36.239,156.823
C03235=1041.759,-18.582,420.615,169.415,36.240,156.823
C03236=1041.765,-18.333,420.602,169.418,36.240,156.823
C03237=1041.771,-18.083,420.588,169.420,36.242,156.823
C03238=1041.778,-17.834,420.574,169.422,36.242,156.823
C03239=1041.784,-17.584,420.560,169.424,36.243,156.824
C03240=1041.790,-17.335,420.546,169.426,36.244,156.824
C03241=1041.796,-17.085,420.532,169.428,36.244,156.824
C03242=1041.802,-16.836,420.518,169.430,36.245,156.824
C03243=1041.810,-16.586,420.504,169.432,36.246,156.824
C03244=1041.816,-16.336,420.490,169.434,36.247,156.824
C03245=1041.822,-16.087,420.476,169.436,36.247,156.824
C03246=1041.828,-15.837,420.461,169.438,36.248,156.825
C03247=1041.835,-15.588,420.447,169.440,36.249,156.825
C03248=1041.841,-15.338,420.433,169.442,36.249,156.825
C03249=1041.847,-15.090,420.419,169.445,36.251,156.825
C03250=1041.853,-14.839,420.405,169.447,36.251,156.825
C03251=1041.861,-14.590,420.391,169.449,36.252,156.825
C03252=1041.866,-14.340,420.377,169.451,36.253,156.825
C03253=1041.872,-14.091,420.362,169.453,36.254,156.826
C03254=1041.879,-13.841,420.349,169.455,36.255,156.826
C03255=1041.885,-13.592,420.334,169.457,36.256,156.826
C03256=1041.891,-13.342,420.320,169.459,36.257,156.826
C03257=1041.898,-13.093,420.305,169.461,36.257,156.826
C03258=1041.904,-12.843,420.290,169.463,36.258,156.826
C03259=1041.909,-12.594,420.277,169.465,36.259,156.826
C03260=1041.917,-12.344,420.262,169.467,36.260,156.827
C03261=1041.922,-12.095,420.248,169.469,36.260,156.827
C03262=1041.928,-11.845,420.233,169.472,36.262,156.827
C03263=1041.936,-11.596,420.219,169.474,36.262,156.827
C03264=1041.941,-11.346,420.205,169.476,36.263,156.827
C03265=1041.947,-11.096,420.190,169.478,36.264,156.827
C03266=1041.955,-10.847,420.176,169.480,36.265,156.827
C03267=1041.960,-10.598,420.162,169.482,36.266,156.828
C03268=1041.966,-10.348,420.147,169.484,36.267,156.828
C03269=1041.973,-10.099,420.133,169.486,36.268,156.828
C03270=1041.979,-9.849,420.119,169.488,36.268,156.828
C03271=1041.985,-9.599,420.104,169.490,36.269,156.828
C03272=1041.991,-9.350,420.089,169.492,36.270,156.828
C03273=1041.998,-9.101,420.075,169.494,36.271,156.828
C03274=1042.004,-8.851,420.061,169.497,36.271,156.829
C03275=1042.010,-8.602,420.046,169.499,36.273,156.829
C03276=1042.017,-8.352,420.032,169.501,36.273,156.829
C03277=1042.024,-8.103,420.017,169.503,36.274,156.829
C03278=1042.030,-7.852,420.003,169.505,36.275,156.829
C03279=1042.036,-7.604,419.989,169.507,36.276,156.829
C03280=1042.043,-7.354,419.974,169.509,36.277,156.829
C03281=1042.049,-7.105,419.959,169.511,36.278,156.830
C03282=1042.055,-6.855,419.945,169.513,36.279,156.830
C03283=1042.062,-6.606,419.931,169.515,36.279,156.830
C03284=1042.068,-6.356,419.916,169.517,36.281,156.830
C03285=1042.074,-6.106,419.901,169.519,36.281,156.830
C03286=1042.081,-5.858,419.887,169.521,36.282,156.830
C03287=1042.087,-5.607,419.872,169.523,36.282,156.831
C03288=1042.093,-5.358,419.858,169.525,36.284,156.831
C03289=1042.099,-5.109,419.843,169.527,36.284,156.831
C03290=1042.106,-4.859,419.829,169.529,36.285,156.831
C03291=1042.113,-4.610,419.814,169.531,36.286,156.831
C03292=1042.119,-4.360,419.799,169.533,36.287,156.831
C03293=1042.126,-4.111,419.784,169.535,36.288,156.831
C03294=1042.132,-3.861,419.771,169.537,36.289,156.832
C03295=1042.139,-3.578,419.753,169.539,36.290,156.832
C03296=1042.147,-3.294,419.737,169.542,36.291,156.832
C03297=1042.153,-3.010,419.720,169.545,36.292,156.832
C03298=1042.160,-2.728,419.703,169.547,36.293,156.832
C03299=1042.167,-2.478,419.688,169.549,36.294,156.833
C03300=1042.173,-2.229,419.673,169.551,36.295,156.833
C03301=1042.179,-1.979,419.658,169.553,36.296,156.833
C03302=1042.185,-1.730,419.643,169.555,36.297,156.833
C03303=1042.192,-1.480,419.628,169.557,36.298,156.833
C03304=1042.198,-1.231,419.614,169.558,36.299,156.833
C03305=1042.204,-0.981,419.599,169.560,36.300,156.834
C03306=1042.210,-0.732,419.584,169.562,36.301,156.834
C03307=1042.217,-0.482,419.569,169.565,36.302,156.834
C03308=1042.222,-0.233,419.554,169.567,36.302,156.834
C03309=1042.229,0.017,419.539,169.569,36.304,156.834
C03310=1042.234,0.267,419.524,169.571,36.304,156.834
C03311=1042.241,0.516,419.509,169.573,36.306,156.835
C03312=1042.247,0.765,419.494,169.575,36.306,156.835
C03313=1042.253,1.015,419.479,169.577,36.308,156.835
C03314=1042.259,1.265,419.464,169.579,36.308,156.835
C03315=1042.266,1.514,419.449,169.581,36.310,156.835
C03316=1042.272,1.763,419.434,169.582,36.310,156.835
C03317=1042.278,2.012,419.419,169.585,36.311,156.836
C03318=1042.285,2.262,419.404,169.587,36.312,156.836
C03319=1042.291,2.511,419.389,169.589,36.313,156.836
C03320=1042.297,2.761,419.374,169.591,36.314,156.836
C03321=1042.304,3.011,419.359,169.593,36.315,156.836
C03322=1042.310,3.260,419.345,169.595,36.316,156.836
C03323=1042.316,3.509,419.329,169.597,36.317,156.837
C03324=1042.323,3.758,419.314,169.599,36.318,156.837
C03325=1042.329,4.008,419.299,169.601,36.319,156.837
C03326=1042.335,4.258,419.284,169.602,36.320,156.837
C03327=1042.341,4.508,419.269,169.604,36.321,156.837
C03328=1042.348,4.757,419.253,169.607,36.322,156.837
C03329=1042.354,5.006,419.238,169.609,36.323,156.838
C03330=1042.361,5.256,419.223,169.611,36.324,156.838
C03331=1042.366,5.505,419.209,169.613,36.325,156.838
C03332=1042.373,5.755,419.194,169.615,36.326,156.838
C03333=1042.379,6.004,419.178,169.617,36.327,156.838
C03334=1042.386,6.253,419.163,169.619,36.328,156.839
C03335=1042.392,6.503,419.148,169.620,36.329,156.839
C03336=1042.399,6.753,419.133,169.622,36.329,156.839
C03337=1042.404,7.002,419.117,169.624,36.331,156.839
C03338=1042.411,7.252,419.102,169.627,36.331,156.839
C03339=1042.417,7.501,419.087,169.629,36.333,156.839
C03340=1042.424,7.750,419.071,169.631,36.333,156.840
C03341=1042.430,8.000,419.057,169.633,36.335,156.840
C03342=1042.436,8.249,419.042,169.635,36.335,156.840
C03343=1042.442,8.499,419.027,169.637,36.337,156.840
C03344=1042.449,8.748,419.011,169.638,36.337,156.840
C03345=1042.456,8.997,418.996,169.640,36.338,156.840
C03346=1042.461,9.247,418.981,169.642,36.339,156.841
C03347=1042.468,9.496,418.965,169.644,36.340,156.841
C03348=1042.474,9.746,418.950,169.646,36.341,156.841
C03349=1042.481,9.995,418.935,169.649,36.342,156.841
C03350=1042.487,10.245,418.920,169.651,36.343,156.841
C03351=1042.494,10.494,418.905,169.653,36.344,156.842
C03352=1042.500,10.743,418.889,169.655,36.345,156.842
C03353=1042.507,10.993,418.874,169.656,36.346,156.842
C03354=1042.513,11.243,418.859,169.658,36.347,156.842
C03355=1042.519,11.492,418.843,169.660,36.347,156.842
C03356=1042.526,11.742,418.828,169.662,36.349,156.842
C03357=1042.532,11.991,418.812,169.664,36.349,156.842
C03358=1042.539,12.240,418.797,169.666,36.351,156.843
C03359=1042.546,12.526,418.780,169.669,36.352,156.843
C03360=1042.554,12.811,418.762,169.671,36.353,156.843
C03361=1042.561,13.096,418.744,169.673,36.354,156.843
C03362=1042.568,13.382,418.727,169.675,36.355,156.843
C03363=1042.574,13.631,418.711,169.677,36.356,156.844
C03364=1042.581,13.881,418.696,169.679,36.357,156.844
C03365=1042.587,14.130,418.680,169.681,36.358,156.844
C03366=1042.594,14.380,418.665,169.683,36.359,156.844
C03367=1042.600,14.629,418.649,169.685,36.360,156.844
C03368=1042.606,14.879,418.634,169.688,36.361,156.844
C03369=1042.613,15.128,418.619,169.689,36.362,156.845
C03370=1042.619,15.377,418.602,169.691,36.363,156.845
C03371=1042.625,15.627,418.587,169.693,36.364,156.845
C03372=1042.631,15.876,418.571,169.695,36.365,156.845
C03373=1042.638,16.126,418.556,169.697,36.366,156.845
C03374=1042.644,16.375,418.541,169.699,36.367,156.846
C03375=1042.650,16.624,418.524,169.700,36.368,156.846
C03376=1042.657,16.874,418.509,169.702,36.369,156.846
C03377=1042.663,17.123,418.493,169.705,36.370,156.846
C03378=1042.669,17.373,418.478,169.707,36.371,156.846
C03379=1042.676,17.622,418.462,169.709,36.372,156.847
C03380=1042.682,17.872,418.446,169.711,36.373,156.847
C03381=1042.689,18.121,418.431,169.712,36.374,156.847
C03382=1042.694,18.371,418.415,169.714,36.376,156.847
C03383=1042.701,18.620,418.399,169.716,36.376,156.847
C03384=1042.708,18.869,418.384,169.718,36.377,156.848
C03385=1042.713,19.119,418.368,169.720,36.378,156.848
C03386=1042.720,19.368,418.352,169.722,36.379,156.848
C03387=1042.726,19.617,418.336,169.724,36.381,156.848
C03388=1042.733,19.867,418.321,169.726,36.381,156.848
C03389=1042.739,20.116,418.305,169.728,36.383,156.848
C03390=1042.746,20.366,418.289,169.730,36.384,156.849
C03391=1042.751,20.616,418.273,169.732,36.384,156.849
C03392=1042.758,20.865,418.257,169.733,36.386,156.849
C03393=1042.764,21.114,418.241,169.735,36.387,156.849
C03394=1042.771,21.363,418.226,169.737,36.388,156.849
C03395=1042.777,21.613,418.209,169.739,36.389,156.850
C03396=1042.783,21.862,418.194,169.742,36.390,156.850
C03397=1042.789,22.112,418.178,169.744,36.391,156.850
C03398=1042.796,22.361,418.162,169.745,36.392,156.850
C03399=1042.802,22.611,418.146,169.747,36.393,156.850
C03400=1042.809,22.860,418.130,169.749,36.394,156.851
C03401=1042.815,23.110,418.115,169.751,36.395,156.851
C03402=1042.821,23.359,418.098,169.753,36.397,156.851
C03403=1042.827,23.608,418.083,169.754,36.397,156.851
C03404=1042.833,23.858,418.066,169.756,36.399,156.851
C03405=1042.840,24.107,418.051,169.759,36.400,156.852
C03406=1042.846,24.357,418.034,169.761,36.400,156.852
C03407=1042.853,24.606,418.018,169.763,36.402,156.852
C03408=1042.859,24.856,418.003,169.764,36.403,156.852
C03409=1042.865,25.105,417.987,169.766,36.404,156.852
C03410=1042.871,25.354,417.971,169.768,36.405,156.852
C03411=1042.878,25.604,417.954,169.770,36.406,156.853
C03412=1042.885,25.853,417.939,169.772,36.407,156.853
C03413=1042.891,26.102,417.922,169.773,36.408,156.853
C03414=1042.897,26.351,417.907,169.776,36.409,156.853
C03415=1042.903,26.601,417.891,169.778,36.410,156.853
C03416=1042.910,26.851,417.874,169.780,36.411,156.854
C03417=1042.916,27.100,417.858,169.782,36.413,156.854
C03418=1042.922,27.349,417.842,169.783,36.413,156.854
C03419=1042.929,27.598,417.826,169.785,36.414,156.854
C03420=1042.935,27.848,417.810,169.787,36.416,156.854
C03421=1042.942,28.098,417.793,169.789,36.417,156.855
C03422=1042.948,28.347,417.778,169.791,36.418,156.855
C03423=1042.955,28.634,417.759,169.794,36.419,156.855
C03424=1042.962,28.920,417.741,169.796,36.420,156.855
C03425=1042.969,29.206,417.722,169.798,36.421,156.856
C03426=1042.977,29.493,417.704,169.800,36.423,156.856
C03427=1042.983,29.743,417.687,169.802,36.424,156.856
C03428=1042.989,29.992,417.670,169.803,36.425,156.856
C03429=1042.995,30.241,417.654,169.805,36.427,156.856
C03430=1043.001,30.491,417.638,169.808,36.427,156.857
C03431=1043.009,30.741,417.622,169.810,36.428,156.857
C03432=1043.014,30.990,417.606,169.811,36.430,156.857
C03433=1043.020,31.239,417.589,169.813,36.431,156.857
C03434=1043.026,31.489,417.573,169.815,36.432,156.857
C03435=1043.033,31.739,417.557,169.817,36.433,156.858
C03436=1043.040,31.987,417.540,169.818,36.434,156.858
C03437=1043.046,32.236,417.524,169.820,36.435,156.858
C03438=1043.052,32.486,417.508,169.822,36.436,156.858
C03439=1043.058,32.736,417.491,169.825,36.437,156.858
C03440=1043.064,32.985,417.475,169.827,36.439,156.859
C03441=1043.071,33.234,417.459,169.828,36.440,156.859
C03442=1043.077,33.484,417.443,169.830,36.440,156.859
C03443=1043.084,33.733,417.426,169.832,36.442,156.859
C03444=1043.090,33.982,417.409,169.834,36.443,156.859
C03445=1043.096,34.232,417.393,169.835,36.444,156.860
C03446=1043.102,34.482,417.376,169.837,36.445,156.860
C03447=1043.109,34.731,417.361,169.840,36.446,156.860
C03448=1043.115,34.979,417.344,169.842,36.447,156.860
C03449=1043.122,35.230,417.327,169.843,36.449,156.861
C03450=1043.128,35.479,417.311,169.845,36.449,156.861
C03451=1043.134,35.728,417.295,169.847,36.451,156.861
C03452=1043.141,35.978,417.277,169.849,36.452,156.861
C03453=1043.147,36.227,417.262,169.851,36.453,156.861
C03454=1043.153,36.476,417.245,169.852,36.454,156.861
C03455=1043.160,36.725,417.228,169.855,36.455,156.862
C03456=1043.166,36.975,417.212,169.857,36.456,156.862
C03457=1043.172,37.224,417.196,169.859,36.458,156.862
C03458=1043.179,37.474,417.179,169.860,36.458,156.862
C03459=1043.185,37.723,417.162,169.862,36.459,156.863
C03460=1043.191,37.972,417.146,169.864,36.461,156.863
C03461=1043.197,38.222,417.129,169.866,36.462,156.863
C03462=1043.204,38.471,417.112,169.867,36.463,156.863
C03463=1043.209,38.720,417.096,169.870,36.465,156.863
C03464=1043.216,38.970,417.079,169.872,36.465,156.864
C03465=1043.222,39.219,417.062,169.874,36.466,156.864
C03466=1043.228,39.469,417.046,169.875,36.468,156.864
C03467=1043.235,39.718,417.029,169.877,36.469,156.864
C03468=1043.241,39.967,417.012,169.879,36.470,156.865
C03469=1043.248,40.217,416.995,169.881,36.472,156.865
C03470=1043.254,40.466,416.979,169.882,36.472,156.865
C03471=1043.260,40.715,416.963,169.885,36.473,156.865
C03472=1043.267,40.965,416.945,169.887,36.475,156.865
C03473=1043.273,41.214,416.929,169.888,36.476,156.866
C03474=1043.279,41.463,416.912,169.890,36.477,156.866
C03475=1043.285,41.713,416.895,169.892,36.478,156.866
C03476=1043.292,41.962,416.878,169.894,36.479,156.866
C03477=1043.297,42.212,416.861,169.895,36.480,156.866
C03478=1043.304,42.461,416.844,169.897,36.482,156.867
C03479=1043.310,42.710,416.828,169.900,36.483,156.867
C03480=1043.317,42.960,416.811,169.902,36.484,156.867
C03481=1043.323,43.209,416.794,169.903,36.485,156.867
C03482=1043.329,43.458,416.777,169.905,36.486,156.867
C03483=1043.335,43.708,416.761,169.907,36.487,156.868
C03484=1043.341,43.957,416.743,169.909,36.489,156.868
C03485=1043.347,44.207,416.727,169.910,36.490,156.868
C03486=1043.354,44.456,416.710,169.912,36.491,156.868
C03487=1043.361,44.743,416.690,169.915,36.493,156.869
C03488=1043.368,45.029,416.670,169.917,36.494,156.869
C03489=1043.375,45.315,416.651,169.919,36.496,156.869
C03490=1043.382,45.602,416.630,169.921,36.497,156.869
C03491=1043.388,45.851,416.614,169.922,36.498,156.870
C03492=1043.394,46.100,416.597,169.924,36.499,156.870
C03493=1043.400,46.350,416.580,169.927,36.501,156.870
C03494=1043.406,46.599,416.563,169.929,36.502,156.870
C03495=1043.413,46.849,416.546,169.930,36.503,156.871
C03496=1043.418,47.098,416.529,169.932,36.504,156.871
C03497=1043.425,47.348,416.511,169.934,36.506,156.871
C03498=1043.432,47.596,416.495,169.935,36.507,156.871
C03499=1043.437,47.845,416.477,169.937,36.508,156.872
C03500=1043.444,48.095,416.460,169.939,36.509,156.872
C03501=1043.450,48.344,416.443,169.942,36.511,156.872
C03502=1043.456,48.594,416.425,169.943,36.512,156.872
C03503=1043.462,48.843,416.409,169.945,36.513,156.873
C03504=1043.469,49.093,416.392,169.947,36.514,156.873
C03505=1043.474,49.342,416.374,169.948,36.516,156.873
C03506=1043.481,49.591,416.357,169.950,36.516,156.873
C03507=1043.487,49.840,416.341,169.952,36.518,156.873
C03508=1043.493,50.090,416.323,169.955,36.519,156.874
C03509=1043.500,50.339,416.306,169.956,36.520,156.874
C03510=1043.506,50.588,416.288,169.958,36.521,156.874
C03511=1043.512,50.838,416.272,169.960,36.523,156.874
C03512=1043.518,51.087,416.254,169.961,36.524,156.875
C03513=1043.525,51.336,416.237,169.963,36.525,156.875
C03514=1043.531,51.586,416.219,169.965,36.526,156.875
C03515=1043.537,51.835,416.202,169.968,36.528,156.875
C03516=1043.543,52.085,416.185,169.969,36.529,156.875
C03517=1043.549,52.334,416.168,169.971,36.530,156.876
C03518=1043.556,52.583,416.151,169.973,36.531,156.876
C03519=1043.562,52.832,416.133,169.974,36.532,156.876
C03520=1043.568,53.082,416.116,169.976,36.533,156.876
C03521=1043.575,53.331,416.099,169.978,36.535,156.877
C03522=1043.580,53.581,416.082,169.979,36.536,156.877
C03523=1043.587,53.830,416.064,169.982,36.537,156.877
C03524=1043.594,54.079,416.047,169.984,36.538,156.877
C03525=1043.600,54.329,416.029,169.986,36.540,156.877
C03526=1043.606,54.577,416.013,169.987,36.541,156.878
C03527=1043.612,54.827,415.995,169.989,36.542,156.878
C03528=1043.619,55.077,415.977,169.991,36.543,156.878
C03529=1043.625,55.325,415.960,169.992,36.544,156.878
C03530=1043.631,55.575,415.942,169.995,36.545,156.879
C03531=1043.638,55.824,415.925,169.997,36.547,156.879
C03532=1043.644,56.074,415.907,169.999,36.548,156.879
C03533=1043.650,56.324,415.891,170.000,36.549,156.879
C03534=1043.656,56.572,415.874,170.002,36.550,156.880
C03535=1043.663,56.822,415.856,170.004,36.552,156.880
C03536=1043.669,57.071,415.839,170.005,36.553,156.880
C03537=1043.676,57.320,415.822,170.008,36.554,156.880
C03538=1043.682,57.570,415.804,170.010,36.555,156.880
C03539=1043.688,57.819,415.787,170.012,36.556,156.881
C03540=1043.694,58.068,415.769,170.013,36.557,156.881
C03541=1043.701,58.318,415.751,170.015,36.559,156.881
C03542=1043.707,58.567,415.734,170.017,36.560,156.881
C03543=1043.713,58.816,415.717,170.018,36.561,156.882
C03544=1043.720,59.066,415.699,170.020,36.562,156.882
C03545=1043.726,59.315,415.682,170.023,36.564,156.882
C03546=1043.733,59.564,415.664,170.025,36.564,156.882
C03547=1043.739,59.814,415.646,170.026,36.565,156.882
C03548=1043.745,60.063,415.629,170.028,36.567,156.883
C03549=1043.752,60.311,415.611,170.030,36.568,156.883
C03550=1043.758,60.561,415.593,170.031,36.569,156.883
C03551=1043.765,60.847,415.573,170.033,36.570,156.883
C03552=1043.773,61.134,415.553,170.036,36.572,156.884
C03553=1043.780,61.420,415.533,170.038,36.573,156.884
C03554=1043.788,61.706,415.513,170.040,36.574,156.884
C03555=1043.794,61.955,415.496,170.042,36.575,156.884
C03556=1043.801,62.205,415.479,170.044,36.577,156.884
C03557=1043.807,62.454,415.461,170.046,36.578,156.885
C03558=1043.814,62.704,415.443,170.047,36.579,156.885
C03559=1043.819,62.952,415.425,170.050,36.580,156.885
C03560=1043.826,63.202,415.408,170.052,36.581,156.885
C03561=1043.833,63.451,415.390,170.053,36.582,156.886
C03562=1043.839,63.701,415.372,170.055,36.584,156.886
C03563=1043.845,63.949,415.355,170.057,36.585,156.886
C03564=1043.852,64.199,415.337,170.059,36.586,156.886
C03565=1043.858,64.448,415.319,170.060,36.587,156.887
C03566=1043.865,64.698,415.301,170.062,36.589,156.887
C03567=1043.870,64.947,415.284,170.065,36.590,156.887
C03568=1043.876,65.197,415.266,170.066,36.591,156.887
C03569=1043.883,65.446,415.247,170.068,36.592,156.887
C03570=1043.889,65.694,415.230,170.070,36.594,156.888
C03571=1043.895,65.944,415.212,170.071,36.595,156.888
C03572=1043.901,66.194,415.194,170.073,36.596,156.888
C03573=1043.909,66.443,415.176,170.075,36.597,156.888
C03574=1043.914,66.692,415.159,170.077,36.599,156.889
C03575=1043.920,66.941,415.141,170.079,36.600,156.889
C03576=1043.927,67.190,415.123,170.081,36.601,156.889
C03577=1043.933,67.440,415.105,170.083,36.602,156.889
C03578=1043.939,67.689,415.087,170.084,36.604,156.890
C03579=1043.945,67.938,415.069,170.086,36.605,156.890
C03580=1043.952,68.188,415.051,170.089,36.606,156.890
C03581=1043.958,68.437,415.033,170.090,36.607,156.890
C03582=1043.964,68.686,415.015,170.092,36.609,156.891
C03583=1043.970,68.936,414.997,170.094,36.610,156.891
C03584=1043.977,69.185,414.980,170.095,36.611,156.891
C03585=1043.984,69.434,414.961,170.097,36.612,156.891
C03586=1043.989,69.683,414.944,170.099,36.614,156.892
C03587=1043.996,69.932,414.925,170.101,36.615,156.892
C03588=1044.002,70.182,414.907,170.103,36.616,156.892
C03589=1044.008,70.431,414.888,170.105,36.617,156.892
C03590=1044.014,70.681,414.871,170.106,36.619,156.892
C03591=1044.020,70.930,414.853,170.108,36.620,156.893
C03592=1044.027,71.179,414.835,170.110,36.621,156.893
C03593=1044.033,71.428,414.817,170.112,36.622,156.893
C03594=1044.039,71.678,414.798,170.114,36.624,156.893
C03595=1044.045,71.927,414.781,170.116,36.625,156.894
C03596=1044.051,72.176,414.762,170.118,36.626,156.894
C03597=1044.058,72.425,414.744,170.119,36.627,156.894
C03598=1044.064,72.675,414.726,170.121,36.629,156.894
C03599=1044.070,72.924,414.708,170.123,36.630,156.895
C03600=1044.076,73.173,414.689,170.124,36.631,156.895
C03601=1044.082,73.422,414.671,170.127,36.632,156.895
C03602=1044.089,73.671,414.653,170.129,36.634,156.895
C03603=1044.096,73.920,414.635,170.130,36.635,156.896
C03604=1044.102,74.170,414.617,170.132,36.636,156.896
C03605=1044.108,74.419,414.598,170.134,36.637,156.896
C03606=1044.114,74.668,414.581,170.135,36.639,156.896
C03607=1044.120,74.917,414.562,170.137,36.640,156.897
C03608=1044.126,75.167,414.544,170.140,36.641,156.897
C03609=1044.133,75.416,414.525,170.141,36.643,156.897
C03610=1044.139,75.665,414.507,170.143,36.644,156.897
C03611=1044.145,75.915,414.489,170.145,36.646,156.898
C03612=1044.152,76.164,414.470,170.147,36.647,156.898
C03613=1044.157,76.413,414.453,170.148,36.648,156.898
C03614=1044.164,76.662,414.434,170.151,36.649,156.898
C03615=1044.171,76.948,414.413,170.153,36.651,156.899
C03616=1044.179,77.235,414.391,170.155,36.652,156.899
C03617=1044.186,77.520,414.371,170.157,36.654,156.899
C03618=1044.193,77.807,414.350,170.159,36.655,156.899
C03619=1044.199,78.056,414.331,170.160,36.656,156.900
C03620=1044.206,78.305,414.312,170.163,36.657,156.900
C03621=1044.211,78.554,414.295,170.165,36.659,156.900
C03622=1044.217,78.803,414.276,170.166,36.660,156.900
C03623=1044.224,79.053,414.257,170.168,36.661,156.901
C03624=1044.230,79.302,414.238,170.170,36.663,156.901
C03625=1044.236,79.552,414.220,170.171,36.664,156.901
C03626=1044.242,79.801,414.202,170.173,36.666,156.901
C03627=1044.249,80.050,414.183,170.176,36.667,156.902
C03628=1044.255,80.299,414.164,170.177,36.668,156.902
C03629=1044.260,80.548,414.145,170.179,36.669,156.902
C03630=1044.266,80.798,414.128,170.181,36.671,156.902
C03631=1044.273,81.047,414.109,170.182,36.672,156.903
C03632=1044.279,81.296,414.090,170.184,36.674,156.903
C03633=1044.285,81.545,414.072,170.187,36.675,156.903
C03634=1044.291,81.794,414.052,170.188,36.676,156.903
C03635=1044.298,82.043,414.034,170.190,36.677,156.904
C03636=1044.304,82.293,414.016,170.192,36.679,156.904
C03637=1044.310,82.542,413.997,170.193,36.680,156.904
C03638=1044.317,82.791,413.978,170.195,36.681,156.904
